    ! ---- P05 weld slots ----
    PERS bool P05W01_Used := FALSE;
    PERS num  P05W01_SubType := 0;
    PERS num  P05W01_ToolSel := 0;
    PERS num  P05W01_LenMM := 0;
    PERS robtarget P05W01_ArcStart := [[0,0,0],[1,0,0,0],[0,0,0,0],[9E9,9E9,9E9,9E9,9E9,9E9]];
    PERS robtarget P05W01_ArcEnd   := [[0,0,0],[1,0,0,0],[0,0,0,0],[9E9,9E9,9E9,9E9,9E9,9E9]];
    PERS robtarget P05W01_Approach := [[0,0,0],[1,0,0,0],[0,0,0,0],[9E9,9E9,9E9,9E9,9E9,9E9]];
    PERS robtarget P05W01_Retract  := [[0,0,0],[1,0,0,0],[0,0,0,0],[9E9,9E9,9E9,9E9,9E9,9E9]];
    PERS robtarget P05W01_Trans    := [[0,0,0],[1,0,0,0],[0,0,0,0],[9E9,9E9,9E9,9E9,9E9,9E9]];
    PERS bool P05W02_Used := FALSE;
    PERS num  P05W02_SubType := 0;
    PERS num  P05W02_ToolSel := 0;
    PERS num  P05W02_LenMM := 0;
    PERS robtarget P05W02_ArcStart := [[0,0,0],[1,0,0,0],[0,0,0,0],[9E9,9E9,9E9,9E9,9E9,9E9]];
    PERS robtarget P05W02_ArcEnd   := [[0,0,0],[1,0,0,0],[0,0,0,0],[9E9,9E9,9E9,9E9,9E9,9E9]];
    PERS robtarget P05W02_Approach := [[0,0,0],[1,0,0,0],[0,0,0,0],[9E9,9E9,9E9,9E9,9E9,9E9]];
    PERS robtarget P05W02_Retract  := [[0,0,0],[1,0,0,0],[0,0,0,0],[9E9,9E9,9E9,9E9,9E9,9E9]];
    PERS robtarget P05W02_Trans    := [[0,0,0],[1,0,0,0],[0,0,0,0],[9E9,9E9,9E9,9E9,9E9,9E9]];
    PERS bool P05W03_Used := FALSE;
    PERS num  P05W03_SubType := 0;
    PERS num  P05W03_ToolSel := 0;
    PERS num  P05W03_LenMM := 0;
    PERS robtarget P05W03_ArcStart := [[0,0,0],[1,0,0,0],[0,0,0,0],[9E9,9E9,9E9,9E9,9E9,9E9]];
    PERS robtarget P05W03_ArcEnd   := [[0,0,0],[1,0,0,0],[0,0,0,0],[9E9,9E9,9E9,9E9,9E9,9E9]];
    PERS robtarget P05W03_Approach := [[0,0,0],[1,0,0,0],[0,0,0,0],[9E9,9E9,9E9,9E9,9E9,9E9]];
    PERS robtarget P05W03_Retract  := [[0,0,0],[1,0,0,0],[0,0,0,0],[9E9,9E9,9E9,9E9,9E9,9E9]];
    PERS robtarget P05W03_Trans    := [[0,0,0],[1,0,0,0],[0,0,0,0],[9E9,9E9,9E9,9E9,9E9,9E9]];
    PERS bool P05W04_Used := FALSE;
    PERS num  P05W04_SubType := 0;
    PERS num  P05W04_ToolSel := 0;
    PERS num  P05W04_LenMM := 0;
    PERS robtarget P05W04_ArcStart := [[0,0,0],[1,0,0,0],[0,0,0,0],[9E9,9E9,9E9,9E9,9E9,9E9]];
    PERS robtarget P05W04_ArcEnd   := [[0,0,0],[1,0,0,0],[0,0,0,0],[9E9,9E9,9E9,9E9,9E9,9E9]];
    PERS robtarget P05W04_Approach := [[0,0,0],[1,0,0,0],[0,0,0,0],[9E9,9E9,9E9,9E9,9E9,9E9]];
    PERS robtarget P05W04_Retract  := [[0,0,0],[1,0,0,0],[0,0,0,0],[9E9,9E9,9E9,9E9,9E9,9E9]];
    PERS robtarget P05W04_Trans    := [[0,0,0],[1,0,0,0],[0,0,0,0],[9E9,9E9,9E9,9E9,9E9,9E9]];
    PERS bool P05W05_Used := FALSE;
    PERS num  P05W05_SubType := 0;
    PERS num  P05W05_ToolSel := 0;
    PERS num  P05W05_LenMM := 0;
    PERS robtarget P05W05_ArcStart := [[0,0,0],[1,0,0,0],[0,0,0,0],[9E9,9E9,9E9,9E9,9E9,9E9]];
    PERS robtarget P05W05_ArcEnd   := [[0,0,0],[1,0,0,0],[0,0,0,0],[9E9,9E9,9E9,9E9,9E9,9E9]];
    PERS robtarget P05W05_Approach := [[0,0,0],[1,0,0,0],[0,0,0,0],[9E9,9E9,9E9,9E9,9E9,9E9]];
    PERS robtarget P05W05_Retract  := [[0,0,0],[1,0,0,0],[0,0,0,0],[9E9,9E9,9E9,9E9,9E9,9E9]];
    PERS robtarget P05W05_Trans    := [[0,0,0],[1,0,0,0],[0,0,0,0],[9E9,9E9,9E9,9E9,9E9,9E9]];
    PERS bool P05W06_Used := FALSE;
    PERS num  P05W06_SubType := 0;
    PERS num  P05W06_ToolSel := 0;
    PERS num  P05W06_LenMM := 0;
    PERS robtarget P05W06_ArcStart := [[0,0,0],[1,0,0,0],[0,0,0,0],[9E9,9E9,9E9,9E9,9E9,9E9]];
    PERS robtarget P05W06_ArcEnd   := [[0,0,0],[1,0,0,0],[0,0,0,0],[9E9,9E9,9E9,9E9,9E9,9E9]];
    PERS robtarget P05W06_Approach := [[0,0,0],[1,0,0,0],[0,0,0,0],[9E9,9E9,9E9,9E9,9E9,9E9]];
    PERS robtarget P05W06_Retract  := [[0,0,0],[1,0,0,0],[0,0,0,0],[9E9,9E9,9E9,9E9,9E9,9E9]];
    PERS robtarget P05W06_Trans    := [[0,0,0],[1,0,0,0],[0,0,0,0],[9E9,9E9,9E9,9E9,9E9,9E9]];
    PERS bool P05W07_Used := FALSE;
    PERS num  P05W07_SubType := 0;
    PERS num  P05W07_ToolSel := 0;
    PERS num  P05W07_LenMM := 0;
    PERS robtarget P05W07_ArcStart := [[0,0,0],[1,0,0,0],[0,0,0,0],[9E9,9E9,9E9,9E9,9E9,9E9]];
    PERS robtarget P05W07_ArcEnd   := [[0,0,0],[1,0,0,0],[0,0,0,0],[9E9,9E9,9E9,9E9,9E9,9E9]];
    PERS robtarget P05W07_Approach := [[0,0,0],[1,0,0,0],[0,0,0,0],[9E9,9E9,9E9,9E9,9E9,9E9]];
    PERS robtarget P05W07_Retract  := [[0,0,0],[1,0,0,0],[0,0,0,0],[9E9,9E9,9E9,9E9,9E9,9E9]];
    PERS robtarget P05W07_Trans    := [[0,0,0],[1,0,0,0],[0,0,0,0],[9E9,9E9,9E9,9E9,9E9,9E9]];
    PERS bool P05W08_Used := FALSE;
    PERS num  P05W08_SubType := 0;
    PERS num  P05W08_ToolSel := 0;
    PERS num  P05W08_LenMM := 0;
    PERS robtarget P05W08_ArcStart := [[0,0,0],[1,0,0,0],[0,0,0,0],[9E9,9E9,9E9,9E9,9E9,9E9]];
    PERS robtarget P05W08_ArcEnd   := [[0,0,0],[1,0,0,0],[0,0,0,0],[9E9,9E9,9E9,9E9,9E9,9E9]];
    PERS robtarget P05W08_Approach := [[0,0,0],[1,0,0,0],[0,0,0,0],[9E9,9E9,9E9,9E9,9E9,9E9]];
    PERS robtarget P05W08_Retract  := [[0,0,0],[1,0,0,0],[0,0,0,0],[9E9,9E9,9E9,9E9,9E9,9E9]];
    PERS robtarget P05W08_Trans    := [[0,0,0],[1,0,0,0],[0,0,0,0],[9E9,9E9,9E9,9E9,9E9,9E9]];
    PERS bool P05W09_Used := FALSE;
    PERS num  P05W09_SubType := 0;
    PERS num  P05W09_ToolSel := 0;
    PERS num  P05W09_LenMM := 0;
    PERS robtarget P05W09_ArcStart := [[0,0,0],[1,0,0,0],[0,0,0,0],[9E9,9E9,9E9,9E9,9E9,9E9]];
    PERS robtarget P05W09_ArcEnd   := [[0,0,0],[1,0,0,0],[0,0,0,0],[9E9,9E9,9E9,9E9,9E9,9E9]];
    PERS robtarget P05W09_Approach := [[0,0,0],[1,0,0,0],[0,0,0,0],[9E9,9E9,9E9,9E9,9E9,9E9]];
    PERS robtarget P05W09_Retract  := [[0,0,0],[1,0,0,0],[0,0,0,0],[9E9,9E9,9E9,9E9,9E9,9E9]];
    PERS robtarget P05W09_Trans    := [[0,0,0],[1,0,0,0],[0,0,0,0],[9E9,9E9,9E9,9E9,9E9,9E9]];
    PERS bool P05W10_Used := FALSE;
    PERS num  P05W10_SubType := 0;
    PERS num  P05W10_ToolSel := 0;
    PERS num  P05W10_LenMM := 0;
    PERS robtarget P05W10_ArcStart := [[0,0,0],[1,0,0,0],[0,0,0,0],[9E9,9E9,9E9,9E9,9E9,9E9]];
    PERS robtarget P05W10_ArcEnd   := [[0,0,0],[1,0,0,0],[0,0,0,0],[9E9,9E9,9E9,9E9,9E9,9E9]];
    PERS robtarget P05W10_Approach := [[0,0,0],[1,0,0,0],[0,0,0,0],[9E9,9E9,9E9,9E9,9E9,9E9]];
    PERS robtarget P05W10_Retract  := [[0,0,0],[1,0,0,0],[0,0,0,0],[9E9,9E9,9E9,9E9,9E9,9E9]];
    PERS robtarget P05W10_Trans    := [[0,0,0],[1,0,0,0],[0,0,0,0],[9E9,9E9,9E9,9E9,9E9,9E9]];
    PERS bool P05W11_Used := FALSE;
    PERS num  P05W11_SubType := 0;
    PERS num  P05W11_ToolSel := 0;
    PERS num  P05W11_LenMM := 0;
    PERS robtarget P05W11_ArcStart := [[0,0,0],[1,0,0,0],[0,0,0,0],[9E9,9E9,9E9,9E9,9E9,9E9]];
    PERS robtarget P05W11_ArcEnd   := [[0,0,0],[1,0,0,0],[0,0,0,0],[9E9,9E9,9E9,9E9,9E9,9E9]];
    PERS robtarget P05W11_Approach := [[0,0,0],[1,0,0,0],[0,0,0,0],[9E9,9E9,9E9,9E9,9E9,9E9]];
    PERS robtarget P05W11_Retract  := [[0,0,0],[1,0,0,0],[0,0,0,0],[9E9,9E9,9E9,9E9,9E9,9E9]];
    PERS robtarget P05W11_Trans    := [[0,0,0],[1,0,0,0],[0,0,0,0],[9E9,9E9,9E9,9E9,9E9,9E9]];
    PERS bool P05W12_Used := FALSE;
    PERS num  P05W12_SubType := 0;
    PERS num  P05W12_ToolSel := 0;
    PERS num  P05W12_LenMM := 0;
    PERS robtarget P05W12_ArcStart := [[0,0,0],[1,0,0,0],[0,0,0,0],[9E9,9E9,9E9,9E9,9E9,9E9]];
    PERS robtarget P05W12_ArcEnd   := [[0,0,0],[1,0,0,0],[0,0,0,0],[9E9,9E9,9E9,9E9,9E9,9E9]];
    PERS robtarget P05W12_Approach := [[0,0,0],[1,0,0,0],[0,0,0,0],[9E9,9E9,9E9,9E9,9E9,9E9]];
    PERS robtarget P05W12_Retract  := [[0,0,0],[1,0,0,0],[0,0,0,0],[9E9,9E9,9E9,9E9,9E9,9E9]];
    PERS robtarget P05W12_Trans    := [[0,0,0],[1,0,0,0],[0,0,0,0],[9E9,9E9,9E9,9E9,9E9,9E9]];
    PERS bool P05W13_Used := FALSE;
    PERS num  P05W13_SubType := 0;
    PERS num  P05W13_ToolSel := 0;
    PERS num  P05W13_LenMM := 0;
    PERS robtarget P05W13_ArcStart := [[0,0,0],[1,0,0,0],[0,0,0,0],[9E9,9E9,9E9,9E9,9E9,9E9]];
    PERS robtarget P05W13_ArcEnd   := [[0,0,0],[1,0,0,0],[0,0,0,0],[9E9,9E9,9E9,9E9,9E9,9E9]];
    PERS robtarget P05W13_Approach := [[0,0,0],[1,0,0,0],[0,0,0,0],[9E9,9E9,9E9,9E9,9E9,9E9]];
    PERS robtarget P05W13_Retract  := [[0,0,0],[1,0,0,0],[0,0,0,0],[9E9,9E9,9E9,9E9,9E9,9E9]];
    PERS robtarget P05W13_Trans    := [[0,0,0],[1,0,0,0],[0,0,0,0],[9E9,9E9,9E9,9E9,9E9,9E9]];
    PERS bool P05W14_Used := FALSE;
    PERS num  P05W14_SubType := 0;
    PERS num  P05W14_ToolSel := 0;
    PERS num  P05W14_LenMM := 0;
    PERS robtarget P05W14_ArcStart := [[0,0,0],[1,0,0,0],[0,0,0,0],[9E9,9E9,9E9,9E9,9E9,9E9]];
    PERS robtarget P05W14_ArcEnd   := [[0,0,0],[1,0,0,0],[0,0,0,0],[9E9,9E9,9E9,9E9,9E9,9E9]];
    PERS robtarget P05W14_Approach := [[0,0,0],[1,0,0,0],[0,0,0,0],[9E9,9E9,9E9,9E9,9E9,9E9]];
    PERS robtarget P05W14_Retract  := [[0,0,0],[1,0,0,0],[0,0,0,0],[9E9,9E9,9E9,9E9,9E9,9E9]];
    PERS robtarget P05W14_Trans    := [[0,0,0],[1,0,0,0],[0,0,0,0],[9E9,9E9,9E9,9E9,9E9,9E9]];
    PERS bool P05W15_Used := FALSE;
    PERS num  P05W15_SubType := 0;
    PERS num  P05W15_ToolSel := 0;
    PERS num  P05W15_LenMM := 0;
    PERS robtarget P05W15_ArcStart := [[0,0,0],[1,0,0,0],[0,0,0,0],[9E9,9E9,9E9,9E9,9E9,9E9]];
    PERS robtarget P05W15_ArcEnd   := [[0,0,0],[1,0,0,0],[0,0,0,0],[9E9,9E9,9E9,9E9,9E9,9E9]];
    PERS robtarget P05W15_Approach := [[0,0,0],[1,0,0,0],[0,0,0,0],[9E9,9E9,9E9,9E9,9E9,9E9]];
    PERS robtarget P05W15_Retract  := [[0,0,0],[1,0,0,0],[0,0,0,0],[9E9,9E9,9E9,9E9,9E9,9E9]];
    PERS robtarget P05W15_Trans    := [[0,0,0],[1,0,0,0],[0,0,0,0],[9E9,9E9,9E9,9E9,9E9,9E9]];
    PERS bool P05W16_Used := FALSE;
    PERS num  P05W16_SubType := 0;
    PERS num  P05W16_ToolSel := 0;
    PERS num  P05W16_LenMM := 0;
    PERS robtarget P05W16_ArcStart := [[0,0,0],[1,0,0,0],[0,0,0,0],[9E9,9E9,9E9,9E9,9E9,9E9]];
    PERS robtarget P05W16_ArcEnd   := [[0,0,0],[1,0,0,0],[0,0,0,0],[9E9,9E9,9E9,9E9,9E9,9E9]];
    PERS robtarget P05W16_Approach := [[0,0,0],[1,0,0,0],[0,0,0,0],[9E9,9E9,9E9,9E9,9E9,9E9]];
    PERS robtarget P05W16_Retract  := [[0,0,0],[1,0,0,0],[0,0,0,0],[9E9,9E9,9E9,9E9,9E9,9E9]];
    PERS robtarget P05W16_Trans    := [[0,0,0],[1,0,0,0],[0,0,0,0],[9E9,9E9,9E9,9E9,9E9,9E9]];
    PERS bool P05W17_Used := FALSE;
    PERS num  P05W17_SubType := 0;
    PERS num  P05W17_ToolSel := 0;
    PERS num  P05W17_LenMM := 0;
    PERS robtarget P05W17_ArcStart := [[0,0,0],[1,0,0,0],[0,0,0,0],[9E9,9E9,9E9,9E9,9E9,9E9]];
    PERS robtarget P05W17_ArcEnd   := [[0,0,0],[1,0,0,0],[0,0,0,0],[9E9,9E9,9E9,9E9,9E9,9E9]];
    PERS robtarget P05W17_Approach := [[0,0,0],[1,0,0,0],[0,0,0,0],[9E9,9E9,9E9,9E9,9E9,9E9]];
    PERS robtarget P05W17_Retract  := [[0,0,0],[1,0,0,0],[0,0,0,0],[9E9,9E9,9E9,9E9,9E9,9E9]];
    PERS robtarget P05W17_Trans    := [[0,0,0],[1,0,0,0],[0,0,0,0],[9E9,9E9,9E9,9E9,9E9,9E9]];
    PERS bool P05W18_Used := FALSE;
    PERS num  P05W18_SubType := 0;
    PERS num  P05W18_ToolSel := 0;
    PERS num  P05W18_LenMM := 0;
    PERS robtarget P05W18_ArcStart := [[0,0,0],[1,0,0,0],[0,0,0,0],[9E9,9E9,9E9,9E9,9E9,9E9]];
    PERS robtarget P05W18_ArcEnd   := [[0,0,0],[1,0,0,0],[0,0,0,0],[9E9,9E9,9E9,9E9,9E9,9E9]];
    PERS robtarget P05W18_Approach := [[0,0,0],[1,0,0,0],[0,0,0,0],[9E9,9E9,9E9,9E9,9E9,9E9]];
    PERS robtarget P05W18_Retract  := [[0,0,0],[1,0,0,0],[0,0,0,0],[9E9,9E9,9E9,9E9,9E9,9E9]];
    PERS robtarget P05W18_Trans    := [[0,0,0],[1,0,0,0],[0,0,0,0],[9E9,9E9,9E9,9E9,9E9,9E9]];
    PERS bool P05W19_Used := FALSE;
    PERS num  P05W19_SubType := 0;
    PERS num  P05W19_ToolSel := 0;
    PERS num  P05W19_LenMM := 0;
    PERS robtarget P05W19_ArcStart := [[0,0,0],[1,0,0,0],[0,0,0,0],[9E9,9E9,9E9,9E9,9E9,9E9]];
    PERS robtarget P05W19_ArcEnd   := [[0,0,0],[1,0,0,0],[0,0,0,0],[9E9,9E9,9E9,9E9,9E9,9E9]];
    PERS robtarget P05W19_Approach := [[0,0,0],[1,0,0,0],[0,0,0,0],[9E9,9E9,9E9,9E9,9E9,9E9]];
    PERS robtarget P05W19_Retract  := [[0,0,0],[1,0,0,0],[0,0,0,0],[9E9,9E9,9E9,9E9,9E9,9E9]];
    PERS robtarget P05W19_Trans    := [[0,0,0],[1,0,0,0],[0,0,0,0],[9E9,9E9,9E9,9E9,9E9,9E9]];
    PERS bool P05W20_Used := FALSE;
    PERS num  P05W20_SubType := 0;
    PERS num  P05W20_ToolSel := 0;
    PERS num  P05W20_LenMM := 0;
    PERS robtarget P05W20_ArcStart := [[0,0,0],[1,0,0,0],[0,0,0,0],[9E9,9E9,9E9,9E9,9E9,9E9]];
    PERS robtarget P05W20_ArcEnd   := [[0,0,0],[1,0,0,0],[0,0,0,0],[9E9,9E9,9E9,9E9,9E9,9E9]];
    PERS robtarget P05W20_Approach := [[0,0,0],[1,0,0,0],[0,0,0,0],[9E9,9E9,9E9,9E9,9E9,9E9]];
    PERS robtarget P05W20_Retract  := [[0,0,0],[1,0,0,0],[0,0,0,0],[9E9,9E9,9E9,9E9,9E9,9E9]];
    PERS robtarget P05W20_Trans    := [[0,0,0],[1,0,0,0],[0,0,0,0],[9E9,9E9,9E9,9E9,9E9,9E9]];
    PERS bool P05W21_Used := FALSE;
    PERS num  P05W21_SubType := 0;
    PERS num  P05W21_ToolSel := 0;
    PERS num  P05W21_LenMM := 0;
    PERS robtarget P05W21_ArcStart := [[0,0,0],[1,0,0,0],[0,0,0,0],[9E9,9E9,9E9,9E9,9E9,9E9]];
    PERS robtarget P05W21_ArcEnd   := [[0,0,0],[1,0,0,0],[0,0,0,0],[9E9,9E9,9E9,9E9,9E9,9E9]];
    PERS robtarget P05W21_Approach := [[0,0,0],[1,0,0,0],[0,0,0,0],[9E9,9E9,9E9,9E9,9E9,9E9]];
    PERS robtarget P05W21_Retract  := [[0,0,0],[1,0,0,0],[0,0,0,0],[9E9,9E9,9E9,9E9,9E9,9E9]];
    PERS robtarget P05W21_Trans    := [[0,0,0],[1,0,0,0],[0,0,0,0],[9E9,9E9,9E9,9E9,9E9,9E9]];
    PERS bool P05W22_Used := FALSE;
    PERS num  P05W22_SubType := 0;
    PERS num  P05W22_ToolSel := 0;
    PERS num  P05W22_LenMM := 0;
    PERS robtarget P05W22_ArcStart := [[0,0,0],[1,0,0,0],[0,0,0,0],[9E9,9E9,9E9,9E9,9E9,9E9]];
    PERS robtarget P05W22_ArcEnd   := [[0,0,0],[1,0,0,0],[0,0,0,0],[9E9,9E9,9E9,9E9,9E9,9E9]];
    PERS robtarget P05W22_Approach := [[0,0,0],[1,0,0,0],[0,0,0,0],[9E9,9E9,9E9,9E9,9E9,9E9]];
    PERS robtarget P05W22_Retract  := [[0,0,0],[1,0,0,0],[0,0,0,0],[9E9,9E9,9E9,9E9,9E9,9E9]];
    PERS robtarget P05W22_Trans    := [[0,0,0],[1,0,0,0],[0,0,0,0],[9E9,9E9,9E9,9E9,9E9,9E9]];
    PERS bool P05W23_Used := FALSE;
    PERS num  P05W23_SubType := 0;
    PERS num  P05W23_ToolSel := 0;
    PERS num  P05W23_LenMM := 0;
    PERS robtarget P05W23_ArcStart := [[0,0,0],[1,0,0,0],[0,0,0,0],[9E9,9E9,9E9,9E9,9E9,9E9]];
    PERS robtarget P05W23_ArcEnd   := [[0,0,0],[1,0,0,0],[0,0,0,0],[9E9,9E9,9E9,9E9,9E9,9E9]];
    PERS robtarget P05W23_Approach := [[0,0,0],[1,0,0,0],[0,0,0,0],[9E9,9E9,9E9,9E9,9E9,9E9]];
    PERS robtarget P05W23_Retract  := [[0,0,0],[1,0,0,0],[0,0,0,0],[9E9,9E9,9E9,9E9,9E9,9E9]];
    PERS robtarget P05W23_Trans    := [[0,0,0],[1,0,0,0],[0,0,0,0],[9E9,9E9,9E9,9E9,9E9,9E9]];
    PERS bool P05W24_Used := FALSE;
    PERS num  P05W24_SubType := 0;
    PERS num  P05W24_ToolSel := 0;
    PERS num  P05W24_LenMM := 0;
    PERS robtarget P05W24_ArcStart := [[0,0,0],[1,0,0,0],[0,0,0,0],[9E9,9E9,9E9,9E9,9E9,9E9]];
    PERS robtarget P05W24_ArcEnd   := [[0,0,0],[1,0,0,0],[0,0,0,0],[9E9,9E9,9E9,9E9,9E9,9E9]];
    PERS robtarget P05W24_Approach := [[0,0,0],[1,0,0,0],[0,0,0,0],[9E9,9E9,9E9,9E9,9E9,9E9]];
    PERS robtarget P05W24_Retract  := [[0,0,0],[1,0,0,0],[0,0,0,0],[9E9,9E9,9E9,9E9,9E9,9E9]];
    PERS robtarget P05W24_Trans    := [[0,0,0],[1,0,0,0],[0,0,0,0],[9E9,9E9,9E9,9E9,9E9,9E9]];
    PERS bool P05W25_Used := FALSE;
    PERS num  P05W25_SubType := 0;
    PERS num  P05W25_ToolSel := 0;
    PERS num  P05W25_LenMM := 0;
    PERS robtarget P05W25_ArcStart := [[0,0,0],[1,0,0,0],[0,0,0,0],[9E9,9E9,9E9,9E9,9E9,9E9]];
    PERS robtarget P05W25_ArcEnd   := [[0,0,0],[1,0,0,0],[0,0,0,0],[9E9,9E9,9E9,9E9,9E9,9E9]];
    PERS robtarget P05W25_Approach := [[0,0,0],[1,0,0,0],[0,0,0,0],[9E9,9E9,9E9,9E9,9E9,9E9]];
    PERS robtarget P05W25_Retract  := [[0,0,0],[1,0,0,0],[0,0,0,0],[9E9,9E9,9E9,9E9,9E9,9E9]];
    PERS robtarget P05W25_Trans    := [[0,0,0],[1,0,0,0],[0,0,0,0],[9E9,9E9,9E9,9E9,9E9,9E9]];
    PERS bool P05W26_Used := FALSE;
    PERS num  P05W26_SubType := 0;
    PERS num  P05W26_ToolSel := 0;
    PERS num  P05W26_LenMM := 0;
    PERS robtarget P05W26_ArcStart := [[0,0,0],[1,0,0,0],[0,0,0,0],[9E9,9E9,9E9,9E9,9E9,9E9]];
    PERS robtarget P05W26_ArcEnd   := [[0,0,0],[1,0,0,0],[0,0,0,0],[9E9,9E9,9E9,9E9,9E9,9E9]];
    PERS robtarget P05W26_Approach := [[0,0,0],[1,0,0,0],[0,0,0,0],[9E9,9E9,9E9,9E9,9E9,9E9]];
    PERS robtarget P05W26_Retract  := [[0,0,0],[1,0,0,0],[0,0,0,0],[9E9,9E9,9E9,9E9,9E9,9E9]];
    PERS robtarget P05W26_Trans    := [[0,0,0],[1,0,0,0],[0,0,0,0],[9E9,9E9,9E9,9E9,9E9,9E9]];
    PERS bool P05W27_Used := FALSE;
    PERS num  P05W27_SubType := 0;
    PERS num  P05W27_ToolSel := 0;
    PERS num  P05W27_LenMM := 0;
    PERS robtarget P05W27_ArcStart := [[0,0,0],[1,0,0,0],[0,0,0,0],[9E9,9E9,9E9,9E9,9E9,9E9]];
    PERS robtarget P05W27_ArcEnd   := [[0,0,0],[1,0,0,0],[0,0,0,0],[9E9,9E9,9E9,9E9,9E9,9E9]];
    PERS robtarget P05W27_Approach := [[0,0,0],[1,0,0,0],[0,0,0,0],[9E9,9E9,9E9,9E9,9E9,9E9]];
    PERS robtarget P05W27_Retract  := [[0,0,0],[1,0,0,0],[0,0,0,0],[9E9,9E9,9E9,9E9,9E9,9E9]];
    PERS robtarget P05W27_Trans    := [[0,0,0],[1,0,0,0],[0,0,0,0],[9E9,9E9,9E9,9E9,9E9,9E9]];
    PERS bool P05W28_Used := FALSE;
    PERS num  P05W28_SubType := 0;
    PERS num  P05W28_ToolSel := 0;
    PERS num  P05W28_LenMM := 0;
    PERS robtarget P05W28_ArcStart := [[0,0,0],[1,0,0,0],[0,0,0,0],[9E9,9E9,9E9,9E9,9E9,9E9]];
    PERS robtarget P05W28_ArcEnd   := [[0,0,0],[1,0,0,0],[0,0,0,0],[9E9,9E9,9E9,9E9,9E9,9E9]];
    PERS robtarget P05W28_Approach := [[0,0,0],[1,0,0,0],[0,0,0,0],[9E9,9E9,9E9,9E9,9E9,9E9]];
    PERS robtarget P05W28_Retract  := [[0,0,0],[1,0,0,0],[0,0,0,0],[9E9,9E9,9E9,9E9,9E9,9E9]];
    PERS robtarget P05W28_Trans    := [[0,0,0],[1,0,0,0],[0,0,0,0],[9E9,9E9,9E9,9E9,9E9,9E9]];
    PERS bool P05W29_Used := FALSE;
    PERS num  P05W29_SubType := 0;
    PERS num  P05W29_ToolSel := 0;
    PERS num  P05W29_LenMM := 0;
    PERS robtarget P05W29_ArcStart := [[0,0,0],[1,0,0,0],[0,0,0,0],[9E9,9E9,9E9,9E9,9E9,9E9]];
    PERS robtarget P05W29_ArcEnd   := [[0,0,0],[1,0,0,0],[0,0,0,0],[9E9,9E9,9E9,9E9,9E9,9E9]];
    PERS robtarget P05W29_Approach := [[0,0,0],[1,0,0,0],[0,0,0,0],[9E9,9E9,9E9,9E9,9E9,9E9]];
    PERS robtarget P05W29_Retract  := [[0,0,0],[1,0,0,0],[0,0,0,0],[9E9,9E9,9E9,9E9,9E9,9E9]];
    PERS robtarget P05W29_Trans    := [[0,0,0],[1,0,0,0],[0,0,0,0],[9E9,9E9,9E9,9E9,9E9,9E9]];
    PERS bool P05W30_Used := FALSE;
    PERS num  P05W30_SubType := 0;
    PERS num  P05W30_ToolSel := 0;
    PERS num  P05W30_LenMM := 0;
    PERS robtarget P05W30_ArcStart := [[0,0,0],[1,0,0,0],[0,0,0,0],[9E9,9E9,9E9,9E9,9E9,9E9]];
    PERS robtarget P05W30_ArcEnd   := [[0,0,0],[1,0,0,0],[0,0,0,0],[9E9,9E9,9E9,9E9,9E9,9E9]];
    PERS robtarget P05W30_Approach := [[0,0,0],[1,0,0,0],[0,0,0,0],[9E9,9E9,9E9,9E9,9E9,9E9]];
    PERS robtarget P05W30_Retract  := [[0,0,0],[1,0,0,0],[0,0,0,0],[9E9,9E9,9E9,9E9,9E9,9E9]];
    PERS robtarget P05W30_Trans    := [[0,0,0],[1,0,0,0],[0,0,0,0],[9E9,9E9,9E9,9E9,9E9,9E9]];

    ! ---- P06 weld slots ----
    PERS bool P06W01_Used := FALSE;
    PERS num  P06W01_SubType := 0;
    PERS num  P06W01_ToolSel := 0;
    PERS num  P06W01_LenMM := 0;
    PERS robtarget P06W01_ArcStart := [[0,0,0],[1,0,0,0],[0,0,0,0],[9E9,9E9,9E9,9E9,9E9,9E9]];
    PERS robtarget P06W01_ArcEnd   := [[0,0,0],[1,0,0,0],[0,0,0,0],[9E9,9E9,9E9,9E9,9E9,9E9]];
    PERS robtarget P06W01_Approach := [[0,0,0],[1,0,0,0],[0,0,0,0],[9E9,9E9,9E9,9E9,9E9,9E9]];
    PERS robtarget P06W01_Retract  := [[0,0,0],[1,0,0,0],[0,0,0,0],[9E9,9E9,9E9,9E9,9E9,9E9]];
    PERS robtarget P06W01_Trans    := [[0,0,0],[1,0,0,0],[0,0,0,0],[9E9,9E9,9E9,9E9,9E9,9E9]];
    PERS bool P06W02_Used := FALSE;
    PERS num  P06W02_SubType := 0;
    PERS num  P06W02_ToolSel := 0;
    PERS num  P06W02_LenMM := 0;
    PERS robtarget P06W02_ArcStart := [[0,0,0],[1,0,0,0],[0,0,0,0],[9E9,9E9,9E9,9E9,9E9,9E9]];
    PERS robtarget P06W02_ArcEnd   := [[0,0,0],[1,0,0,0],[0,0,0,0],[9E9,9E9,9E9,9E9,9E9,9E9]];
    PERS robtarget P06W02_Approach := [[0,0,0],[1,0,0,0],[0,0,0,0],[9E9,9E9,9E9,9E9,9E9,9E9]];
    PERS robtarget P06W02_Retract  := [[0,0,0],[1,0,0,0],[0,0,0,0],[9E9,9E9,9E9,9E9,9E9,9E9]];
    PERS robtarget P06W02_Trans    := [[0,0,0],[1,0,0,0],[0,0,0,0],[9E9,9E9,9E9,9E9,9E9,9E9]];
    PERS bool P06W03_Used := FALSE;
    PERS num  P06W03_SubType := 0;
    PERS num  P06W03_ToolSel := 0;
    PERS num  P06W03_LenMM := 0;
    PERS robtarget P06W03_ArcStart := [[0,0,0],[1,0,0,0],[0,0,0,0],[9E9,9E9,9E9,9E9,9E9,9E9]];
    PERS robtarget P06W03_ArcEnd   := [[0,0,0],[1,0,0,0],[0,0,0,0],[9E9,9E9,9E9,9E9,9E9,9E9]];
    PERS robtarget P06W03_Approach := [[0,0,0],[1,0,0,0],[0,0,0,0],[9E9,9E9,9E9,9E9,9E9,9E9]];
    PERS robtarget P06W03_Retract  := [[0,0,0],[1,0,0,0],[0,0,0,0],[9E9,9E9,9E9,9E9,9E9,9E9]];
    PERS robtarget P06W03_Trans    := [[0,0,0],[1,0,0,0],[0,0,0,0],[9E9,9E9,9E9,9E9,9E9,9E9]];
    PERS bool P06W04_Used := FALSE;
    PERS num  P06W04_SubType := 0;
    PERS num  P06W04_ToolSel := 0;
    PERS num  P06W04_LenMM := 0;
    PERS robtarget P06W04_ArcStart := [[0,0,0],[1,0,0,0],[0,0,0,0],[9E9,9E9,9E9,9E9,9E9,9E9]];
    PERS robtarget P06W04_ArcEnd   := [[0,0,0],[1,0,0,0],[0,0,0,0],[9E9,9E9,9E9,9E9,9E9,9E9]];
    PERS robtarget P06W04_Approach := [[0,0,0],[1,0,0,0],[0,0,0,0],[9E9,9E9,9E9,9E9,9E9,9E9]];
    PERS robtarget P06W04_Retract  := [[0,0,0],[1,0,0,0],[0,0,0,0],[9E9,9E9,9E9,9E9,9E9,9E9]];
    PERS robtarget P06W04_Trans    := [[0,0,0],[1,0,0,0],[0,0,0,0],[9E9,9E9,9E9,9E9,9E9,9E9]];
    PERS bool P06W05_Used := FALSE;
    PERS num  P06W05_SubType := 0;
    PERS num  P06W05_ToolSel := 0;
    PERS num  P06W05_LenMM := 0;
    PERS robtarget P06W05_ArcStart := [[0,0,0],[1,0,0,0],[0,0,0,0],[9E9,9E9,9E9,9E9,9E9,9E9]];
    PERS robtarget P06W05_ArcEnd   := [[0,0,0],[1,0,0,0],[0,0,0,0],[9E9,9E9,9E9,9E9,9E9,9E9]];
    PERS robtarget P06W05_Approach := [[0,0,0],[1,0,0,0],[0,0,0,0],[9E9,9E9,9E9,9E9,9E9,9E9]];
    PERS robtarget P06W05_Retract  := [[0,0,0],[1,0,0,0],[0,0,0,0],[9E9,9E9,9E9,9E9,9E9,9E9]];
    PERS robtarget P06W05_Trans    := [[0,0,0],[1,0,0,0],[0,0,0,0],[9E9,9E9,9E9,9E9,9E9,9E9]];
    PERS bool P06W06_Used := FALSE;
    PERS num  P06W06_SubType := 0;
    PERS num  P06W06_ToolSel := 0;
    PERS num  P06W06_LenMM := 0;
    PERS robtarget P06W06_ArcStart := [[0,0,0],[1,0,0,0],[0,0,0,0],[9E9,9E9,9E9,9E9,9E9,9E9]];
    PERS robtarget P06W06_ArcEnd   := [[0,0,0],[1,0,0,0],[0,0,0,0],[9E9,9E9,9E9,9E9,9E9,9E9]];
    PERS robtarget P06W06_Approach := [[0,0,0],[1,0,0,0],[0,0,0,0],[9E9,9E9,9E9,9E9,9E9,9E9]];
    PERS robtarget P06W06_Retract  := [[0,0,0],[1,0,0,0],[0,0,0,0],[9E9,9E9,9E9,9E9,9E9,9E9]];
    PERS robtarget P06W06_Trans    := [[0,0,0],[1,0,0,0],[0,0,0,0],[9E9,9E9,9E9,9E9,9E9,9E9]];
    PERS bool P06W07_Used := FALSE;
    PERS num  P06W07_SubType := 0;
    PERS num  P06W07_ToolSel := 0;
    PERS num  P06W07_LenMM := 0;
    PERS robtarget P06W07_ArcStart := [[0,0,0],[1,0,0,0],[0,0,0,0],[9E9,9E9,9E9,9E9,9E9,9E9]];
    PERS robtarget P06W07_ArcEnd   := [[0,0,0],[1,0,0,0],[0,0,0,0],[9E9,9E9,9E9,9E9,9E9,9E9]];
    PERS robtarget P06W07_Approach := [[0,0,0],[1,0,0,0],[0,0,0,0],[9E9,9E9,9E9,9E9,9E9,9E9]];
    PERS robtarget P06W07_Retract  := [[0,0,0],[1,0,0,0],[0,0,0,0],[9E9,9E9,9E9,9E9,9E9,9E9]];
    PERS robtarget P06W07_Trans    := [[0,0,0],[1,0,0,0],[0,0,0,0],[9E9,9E9,9E9,9E9,9E9,9E9]];
    PERS bool P06W08_Used := FALSE;
    PERS num  P06W08_SubType := 0;
    PERS num  P06W08_ToolSel := 0;
    PERS num  P06W08_LenMM := 0;
    PERS robtarget P06W08_ArcStart := [[0,0,0],[1,0,0,0],[0,0,0,0],[9E9,9E9,9E9,9E9,9E9,9E9]];
    PERS robtarget P06W08_ArcEnd   := [[0,0,0],[1,0,0,0],[0,0,0,0],[9E9,9E9,9E9,9E9,9E9,9E9]];
    PERS robtarget P06W08_Approach := [[0,0,0],[1,0,0,0],[0,0,0,0],[9E9,9E9,9E9,9E9,9E9,9E9]];
    PERS robtarget P06W08_Retract  := [[0,0,0],[1,0,0,0],[0,0,0,0],[9E9,9E9,9E9,9E9,9E9,9E9]];
    PERS robtarget P06W08_Trans    := [[0,0,0],[1,0,0,0],[0,0,0,0],[9E9,9E9,9E9,9E9,9E9,9E9]];
    PERS bool P06W09_Used := FALSE;
    PERS num  P06W09_SubType := 0;
    PERS num  P06W09_ToolSel := 0;
    PERS num  P06W09_LenMM := 0;
    PERS robtarget P06W09_ArcStart := [[0,0,0],[1,0,0,0],[0,0,0,0],[9E9,9E9,9E9,9E9,9E9,9E9]];
    PERS robtarget P06W09_ArcEnd   := [[0,0,0],[1,0,0,0],[0,0,0,0],[9E9,9E9,9E9,9E9,9E9,9E9]];
    PERS robtarget P06W09_Approach := [[0,0,0],[1,0,0,0],[0,0,0,0],[9E9,9E9,9E9,9E9,9E9,9E9]];
    PERS robtarget P06W09_Retract  := [[0,0,0],[1,0,0,0],[0,0,0,0],[9E9,9E9,9E9,9E9,9E9,9E9]];
    PERS robtarget P06W09_Trans    := [[0,0,0],[1,0,0,0],[0,0,0,0],[9E9,9E9,9E9,9E9,9E9,9E9]];
    PERS bool P06W10_Used := FALSE;
    PERS num  P06W10_SubType := 0;
    PERS num  P06W10_ToolSel := 0;
    PERS num  P06W10_LenMM := 0;
    PERS robtarget P06W10_ArcStart := [[0,0,0],[1,0,0,0],[0,0,0,0],[9E9,9E9,9E9,9E9,9E9,9E9]];
    PERS robtarget P06W10_ArcEnd   := [[0,0,0],[1,0,0,0],[0,0,0,0],[9E9,9E9,9E9,9E9,9E9,9E9]];
    PERS robtarget P06W10_Approach := [[0,0,0],[1,0,0,0],[0,0,0,0],[9E9,9E9,9E9,9E9,9E9,9E9]];
    PERS robtarget P06W10_Retract  := [[0,0,0],[1,0,0,0],[0,0,0,0],[9E9,9E9,9E9,9E9,9E9,9E9]];
    PERS robtarget P06W10_Trans    := [[0,0,0],[1,0,0,0],[0,0,0,0],[9E9,9E9,9E9,9E9,9E9,9E9]];
    PERS bool P06W11_Used := FALSE;
    PERS num  P06W11_SubType := 0;
    PERS num  P06W11_ToolSel := 0;
    PERS num  P06W11_LenMM := 0;
    PERS robtarget P06W11_ArcStart := [[0,0,0],[1,0,0,0],[0,0,0,0],[9E9,9E9,9E9,9E9,9E9,9E9]];
    PERS robtarget P06W11_ArcEnd   := [[0,0,0],[1,0,0,0],[0,0,0,0],[9E9,9E9,9E9,9E9,9E9,9E9]];
    PERS robtarget P06W11_Approach := [[0,0,0],[1,0,0,0],[0,0,0,0],[9E9,9E9,9E9,9E9,9E9,9E9]];
    PERS robtarget P06W11_Retract  := [[0,0,0],[1,0,0,0],[0,0,0,0],[9E9,9E9,9E9,9E9,9E9,9E9]];
    PERS robtarget P06W11_Trans    := [[0,0,0],[1,0,0,0],[0,0,0,0],[9E9,9E9,9E9,9E9,9E9,9E9]];
    PERS bool P06W12_Used := FALSE;
    PERS num  P06W12_SubType := 0;
    PERS num  P06W12_ToolSel := 0;
    PERS num  P06W12_LenMM := 0;
    PERS robtarget P06W12_ArcStart := [[0,0,0],[1,0,0,0],[0,0,0,0],[9E9,9E9,9E9,9E9,9E9,9E9]];
    PERS robtarget P06W12_ArcEnd   := [[0,0,0],[1,0,0,0],[0,0,0,0],[9E9,9E9,9E9,9E9,9E9,9E9]];
    PERS robtarget P06W12_Approach := [[0,0,0],[1,0,0,0],[0,0,0,0],[9E9,9E9,9E9,9E9,9E9,9E9]];
    PERS robtarget P06W12_Retract  := [[0,0,0],[1,0,0,0],[0,0,0,0],[9E9,9E9,9E9,9E9,9E9,9E9]];
    PERS robtarget P06W12_Trans    := [[0,0,0],[1,0,0,0],[0,0,0,0],[9E9,9E9,9E9,9E9,9E9,9E9]];
    PERS bool P06W13_Used := FALSE;
    PERS num  P06W13_SubType := 0;
    PERS num  P06W13_ToolSel := 0;
    PERS num  P06W13_LenMM := 0;
    PERS robtarget P06W13_ArcStart := [[0,0,0],[1,0,0,0],[0,0,0,0],[9E9,9E9,9E9,9E9,9E9,9E9]];
    PERS robtarget P06W13_ArcEnd   := [[0,0,0],[1,0,0,0],[0,0,0,0],[9E9,9E9,9E9,9E9,9E9,9E9]];
    PERS robtarget P06W13_Approach := [[0,0,0],[1,0,0,0],[0,0,0,0],[9E9,9E9,9E9,9E9,9E9,9E9]];
    PERS robtarget P06W13_Retract  := [[0,0,0],[1,0,0,0],[0,0,0,0],[9E9,9E9,9E9,9E9,9E9,9E9]];
    PERS robtarget P06W13_Trans    := [[0,0,0],[1,0,0,0],[0,0,0,0],[9E9,9E9,9E9,9E9,9E9,9E9]];
    PERS bool P06W14_Used := FALSE;
    PERS num  P06W14_SubType := 0;
    PERS num  P06W14_ToolSel := 0;
    PERS num  P06W14_LenMM := 0;
    PERS robtarget P06W14_ArcStart := [[0,0,0],[1,0,0,0],[0,0,0,0],[9E9,9E9,9E9,9E9,9E9,9E9]];
    PERS robtarget P06W14_ArcEnd   := [[0,0,0],[1,0,0,0],[0,0,0,0],[9E9,9E9,9E9,9E9,9E9,9E9]];
    PERS robtarget P06W14_Approach := [[0,0,0],[1,0,0,0],[0,0,0,0],[9E9,9E9,9E9,9E9,9E9,9E9]];
    PERS robtarget P06W14_Retract  := [[0,0,0],[1,0,0,0],[0,0,0,0],[9E9,9E9,9E9,9E9,9E9,9E9]];
    PERS robtarget P06W14_Trans    := [[0,0,0],[1,0,0,0],[0,0,0,0],[9E9,9E9,9E9,9E9,9E9,9E9]];
    PERS bool P06W15_Used := FALSE;
    PERS num  P06W15_SubType := 0;
    PERS num  P06W15_ToolSel := 0;
    PERS num  P06W15_LenMM := 0;
    PERS robtarget P06W15_ArcStart := [[0,0,0],[1,0,0,0],[0,0,0,0],[9E9,9E9,9E9,9E9,9E9,9E9]];
    PERS robtarget P06W15_ArcEnd   := [[0,0,0],[1,0,0,0],[0,0,0,0],[9E9,9E9,9E9,9E9,9E9,9E9]];
    PERS robtarget P06W15_Approach := [[0,0,0],[1,0,0,0],[0,0,0,0],[9E9,9E9,9E9,9E9,9E9,9E9]];
    PERS robtarget P06W15_Retract  := [[0,0,0],[1,0,0,0],[0,0,0,0],[9E9,9E9,9E9,9E9,9E9,9E9]];
    PERS robtarget P06W15_Trans    := [[0,0,0],[1,0,0,0],[0,0,0,0],[9E9,9E9,9E9,9E9,9E9,9E9]];
    PERS bool P06W16_Used := FALSE;
    PERS num  P06W16_SubType := 0;
    PERS num  P06W16_ToolSel := 0;
    PERS num  P06W16_LenMM := 0;
    PERS robtarget P06W16_ArcStart := [[0,0,0],[1,0,0,0],[0,0,0,0],[9E9,9E9,9E9,9E9,9E9,9E9]];
    PERS robtarget P06W16_ArcEnd   := [[0,0,0],[1,0,0,0],[0,0,0,0],[9E9,9E9,9E9,9E9,9E9,9E9]];
    PERS robtarget P06W16_Approach := [[0,0,0],[1,0,0,0],[0,0,0,0],[9E9,9E9,9E9,9E9,9E9,9E9]];
    PERS robtarget P06W16_Retract  := [[0,0,0],[1,0,0,0],[0,0,0,0],[9E9,9E9,9E9,9E9,9E9,9E9]];
    PERS robtarget P06W16_Trans    := [[0,0,0],[1,0,0,0],[0,0,0,0],[9E9,9E9,9E9,9E9,9E9,9E9]];
    PERS bool P06W17_Used := FALSE;
    PERS num  P06W17_SubType := 0;
    PERS num  P06W17_ToolSel := 0;
    PERS num  P06W17_LenMM := 0;
    PERS robtarget P06W17_ArcStart := [[0,0,0],[1,0,0,0],[0,0,0,0],[9E9,9E9,9E9,9E9,9E9,9E9]];
    PERS robtarget P06W17_ArcEnd   := [[0,0,0],[1,0,0,0],[0,0,0,0],[9E9,9E9,9E9,9E9,9E9,9E9]];
    PERS robtarget P06W17_Approach := [[0,0,0],[1,0,0,0],[0,0,0,0],[9E9,9E9,9E9,9E9,9E9,9E9]];
    PERS robtarget P06W17_Retract  := [[0,0,0],[1,0,0,0],[0,0,0,0],[9E9,9E9,9E9,9E9,9E9,9E9]];
    PERS robtarget P06W17_Trans    := [[0,0,0],[1,0,0,0],[0,0,0,0],[9E9,9E9,9E9,9E9,9E9,9E9]];
    PERS bool P06W18_Used := FALSE;
    PERS num  P06W18_SubType := 0;
    PERS num  P06W18_ToolSel := 0;
    PERS num  P06W18_LenMM := 0;
    PERS robtarget P06W18_ArcStart := [[0,0,0],[1,0,0,0],[0,0,0,0],[9E9,9E9,9E9,9E9,9E9,9E9]];
    PERS robtarget P06W18_ArcEnd   := [[0,0,0],[1,0,0,0],[0,0,0,0],[9E9,9E9,9E9,9E9,9E9,9E9]];
    PERS robtarget P06W18_Approach := [[0,0,0],[1,0,0,0],[0,0,0,0],[9E9,9E9,9E9,9E9,9E9,9E9]];
    PERS robtarget P06W18_Retract  := [[0,0,0],[1,0,0,0],[0,0,0,0],[9E9,9E9,9E9,9E9,9E9,9E9]];
    PERS robtarget P06W18_Trans    := [[0,0,0],[1,0,0,0],[0,0,0,0],[9E9,9E9,9E9,9E9,9E9,9E9]];
    PERS bool P06W19_Used := FALSE;
    PERS num  P06W19_SubType := 0;
    PERS num  P06W19_ToolSel := 0;
    PERS num  P06W19_LenMM := 0;
    PERS robtarget P06W19_ArcStart := [[0,0,0],[1,0,0,0],[0,0,0,0],[9E9,9E9,9E9,9E9,9E9,9E9]];
    PERS robtarget P06W19_ArcEnd   := [[0,0,0],[1,0,0,0],[0,0,0,0],[9E9,9E9,9E9,9E9,9E9,9E9]];
    PERS robtarget P06W19_Approach := [[0,0,0],[1,0,0,0],[0,0,0,0],[9E9,9E9,9E9,9E9,9E9,9E9]];
    PERS robtarget P06W19_Retract  := [[0,0,0],[1,0,0,0],[0,0,0,0],[9E9,9E9,9E9,9E9,9E9,9E9]];
    PERS robtarget P06W19_Trans    := [[0,0,0],[1,0,0,0],[0,0,0,0],[9E9,9E9,9E9,9E9,9E9,9E9]];
    PERS bool P06W20_Used := FALSE;
    PERS num  P06W20_SubType := 0;
    PERS num  P06W20_ToolSel := 0;
    PERS num  P06W20_LenMM := 0;
    PERS robtarget P06W20_ArcStart := [[0,0,0],[1,0,0,0],[0,0,0,0],[9E9,9E9,9E9,9E9,9E9,9E9]];
    PERS robtarget P06W20_ArcEnd   := [[0,0,0],[1,0,0,0],[0,0,0,0],[9E9,9E9,9E9,9E9,9E9,9E9]];
    PERS robtarget P06W20_Approach := [[0,0,0],[1,0,0,0],[0,0,0,0],[9E9,9E9,9E9,9E9,9E9,9E9]];
    PERS robtarget P06W20_Retract  := [[0,0,0],[1,0,0,0],[0,0,0,0],[9E9,9E9,9E9,9E9,9E9,9E9]];
    PERS robtarget P06W20_Trans    := [[0,0,0],[1,0,0,0],[0,0,0,0],[9E9,9E9,9E9,9E9,9E9,9E9]];
    PERS bool P06W21_Used := FALSE;
    PERS num  P06W21_SubType := 0;
    PERS num  P06W21_ToolSel := 0;
    PERS num  P06W21_LenMM := 0;
    PERS robtarget P06W21_ArcStart := [[0,0,0],[1,0,0,0],[0,0,0,0],[9E9,9E9,9E9,9E9,9E9,9E9]];
    PERS robtarget P06W21_ArcEnd   := [[0,0,0],[1,0,0,0],[0,0,0,0],[9E9,9E9,9E9,9E9,9E9,9E9]];
    PERS robtarget P06W21_Approach := [[0,0,0],[1,0,0,0],[0,0,0,0],[9E9,9E9,9E9,9E9,9E9,9E9]];
    PERS robtarget P06W21_Retract  := [[0,0,0],[1,0,0,0],[0,0,0,0],[9E9,9E9,9E9,9E9,9E9,9E9]];
    PERS robtarget P06W21_Trans    := [[0,0,0],[1,0,0,0],[0,0,0,0],[9E9,9E9,9E9,9E9,9E9,9E9]];
    PERS bool P06W22_Used := FALSE;
    PERS num  P06W22_SubType := 0;
    PERS num  P06W22_ToolSel := 0;
    PERS num  P06W22_LenMM := 0;
    PERS robtarget P06W22_ArcStart := [[0,0,0],[1,0,0,0],[0,0,0,0],[9E9,9E9,9E9,9E9,9E9,9E9]];
    PERS robtarget P06W22_ArcEnd   := [[0,0,0],[1,0,0,0],[0,0,0,0],[9E9,9E9,9E9,9E9,9E9,9E9]];
    PERS robtarget P06W22_Approach := [[0,0,0],[1,0,0,0],[0,0,0,0],[9E9,9E9,9E9,9E9,9E9,9E9]];
    PERS robtarget P06W22_Retract  := [[0,0,0],[1,0,0,0],[0,0,0,0],[9E9,9E9,9E9,9E9,9E9,9E9]];
    PERS robtarget P06W22_Trans    := [[0,0,0],[1,0,0,0],[0,0,0,0],[9E9,9E9,9E9,9E9,9E9,9E9]];
    PERS bool P06W23_Used := FALSE;
    PERS num  P06W23_SubType := 0;
    PERS num  P06W23_ToolSel := 0;
    PERS num  P06W23_LenMM := 0;
    PERS robtarget P06W23_ArcStart := [[0,0,0],[1,0,0,0],[0,0,0,0],[9E9,9E9,9E9,9E9,9E9,9E9]];
    PERS robtarget P06W23_ArcEnd   := [[0,0,0],[1,0,0,0],[0,0,0,0],[9E9,9E9,9E9,9E9,9E9,9E9]];
    PERS robtarget P06W23_Approach := [[0,0,0],[1,0,0,0],[0,0,0,0],[9E9,9E9,9E9,9E9,9E9,9E9]];
    PERS robtarget P06W23_Retract  := [[0,0,0],[1,0,0,0],[0,0,0,0],[9E9,9E9,9E9,9E9,9E9,9E9]];
    PERS robtarget P06W23_Trans    := [[0,0,0],[1,0,0,0],[0,0,0,0],[9E9,9E9,9E9,9E9,9E9,9E9]];
    PERS bool P06W24_Used := FALSE;
    PERS num  P06W24_SubType := 0;
    PERS num  P06W24_ToolSel := 0;
    PERS num  P06W24_LenMM := 0;
    PERS robtarget P06W24_ArcStart := [[0,0,0],[1,0,0,0],[0,0,0,0],[9E9,9E9,9E9,9E9,9E9,9E9]];
    PERS robtarget P06W24_ArcEnd   := [[0,0,0],[1,0,0,0],[0,0,0,0],[9E9,9E9,9E9,9E9,9E9,9E9]];
    PERS robtarget P06W24_Approach := [[0,0,0],[1,0,0,0],[0,0,0,0],[9E9,9E9,9E9,9E9,9E9,9E9]];
    PERS robtarget P06W24_Retract  := [[0,0,0],[1,0,0,0],[0,0,0,0],[9E9,9E9,9E9,9E9,9E9,9E9]];
    PERS robtarget P06W24_Trans    := [[0,0,0],[1,0,0,0],[0,0,0,0],[9E9,9E9,9E9,9E9,9E9,9E9]];
    PERS bool P06W25_Used := FALSE;
    PERS num  P06W25_SubType := 0;
    PERS num  P06W25_ToolSel := 0;
    PERS num  P06W25_LenMM := 0;
    PERS robtarget P06W25_ArcStart := [[0,0,0],[1,0,0,0],[0,0,0,0],[9E9,9E9,9E9,9E9,9E9,9E9]];
    PERS robtarget P06W25_ArcEnd   := [[0,0,0],[1,0,0,0],[0,0,0,0],[9E9,9E9,9E9,9E9,9E9,9E9]];
    PERS robtarget P06W25_Approach := [[0,0,0],[1,0,0,0],[0,0,0,0],[9E9,9E9,9E9,9E9,9E9,9E9]];
    PERS robtarget P06W25_Retract  := [[0,0,0],[1,0,0,0],[0,0,0,0],[9E9,9E9,9E9,9E9,9E9,9E9]];
    PERS robtarget P06W25_Trans    := [[0,0,0],[1,0,0,0],[0,0,0,0],[9E9,9E9,9E9,9E9,9E9,9E9]];
    PERS bool P06W26_Used := FALSE;
    PERS num  P06W26_SubType := 0;
    PERS num  P06W26_ToolSel := 0;
    PERS num  P06W26_LenMM := 0;
    PERS robtarget P06W26_ArcStart := [[0,0,0],[1,0,0,0],[0,0,0,0],[9E9,9E9,9E9,9E9,9E9,9E9]];
    PERS robtarget P06W26_ArcEnd   := [[0,0,0],[1,0,0,0],[0,0,0,0],[9E9,9E9,9E9,9E9,9E9,9E9]];
    PERS robtarget P06W26_Approach := [[0,0,0],[1,0,0,0],[0,0,0,0],[9E9,9E9,9E9,9E9,9E9,9E9]];
    PERS robtarget P06W26_Retract  := [[0,0,0],[1,0,0,0],[0,0,0,0],[9E9,9E9,9E9,9E9,9E9,9E9]];
    PERS robtarget P06W26_Trans    := [[0,0,0],[1,0,0,0],[0,0,0,0],[9E9,9E9,9E9,9E9,9E9,9E9]];
    PERS bool P06W27_Used := FALSE;
    PERS num  P06W27_SubType := 0;
    PERS num  P06W27_ToolSel := 0;
    PERS num  P06W27_LenMM := 0;
    PERS robtarget P06W27_ArcStart := [[0,0,0],[1,0,0,0],[0,0,0,0],[9E9,9E9,9E9,9E9,9E9,9E9]];
    PERS robtarget P06W27_ArcEnd   := [[0,0,0],[1,0,0,0],[0,0,0,0],[9E9,9E9,9E9,9E9,9E9,9E9]];
    PERS robtarget P06W27_Approach := [[0,0,0],[1,0,0,0],[0,0,0,0],[9E9,9E9,9E9,9E9,9E9,9E9]];
    PERS robtarget P06W27_Retract  := [[0,0,0],[1,0,0,0],[0,0,0,0],[9E9,9E9,9E9,9E9,9E9,9E9]];
    PERS robtarget P06W27_Trans    := [[0,0,0],[1,0,0,0],[0,0,0,0],[9E9,9E9,9E9,9E9,9E9,9E9]];
    PERS bool P06W28_Used := FALSE;
    PERS num  P06W28_SubType := 0;
    PERS num  P06W28_ToolSel := 0;
    PERS num  P06W28_LenMM := 0;
    PERS robtarget P06W28_ArcStart := [[0,0,0],[1,0,0,0],[0,0,0,0],[9E9,9E9,9E9,9E9,9E9,9E9]];
    PERS robtarget P06W28_ArcEnd   := [[0,0,0],[1,0,0,0],[0,0,0,0],[9E9,9E9,9E9,9E9,9E9,9E9]];
    PERS robtarget P06W28_Approach := [[0,0,0],[1,0,0,0],[0,0,0,0],[9E9,9E9,9E9,9E9,9E9,9E9]];
    PERS robtarget P06W28_Retract  := [[0,0,0],[1,0,0,0],[0,0,0,0],[9E9,9E9,9E9,9E9,9E9,9E9]];
    PERS robtarget P06W28_Trans    := [[0,0,0],[1,0,0,0],[0,0,0,0],[9E9,9E9,9E9,9E9,9E9,9E9]];
    PERS bool P06W29_Used := FALSE;
    PERS num  P06W29_SubType := 0;
    PERS num  P06W29_ToolSel := 0;
    PERS num  P06W29_LenMM := 0;
    PERS robtarget P06W29_ArcStart := [[0,0,0],[1,0,0,0],[0,0,0,0],[9E9,9E9,9E9,9E9,9E9,9E9]];
    PERS robtarget P06W29_ArcEnd   := [[0,0,0],[1,0,0,0],[0,0,0,0],[9E9,9E9,9E9,9E9,9E9,9E9]];
    PERS robtarget P06W29_Approach := [[0,0,0],[1,0,0,0],[0,0,0,0],[9E9,9E9,9E9,9E9,9E9,9E9]];
    PERS robtarget P06W29_Retract  := [[0,0,0],[1,0,0,0],[0,0,0,0],[9E9,9E9,9E9,9E9,9E9,9E9]];
    PERS robtarget P06W29_Trans    := [[0,0,0],[1,0,0,0],[0,0,0,0],[9E9,9E9,9E9,9E9,9E9,9E9]];
    PERS bool P06W30_Used := FALSE;
    PERS num  P06W30_SubType := 0;
    PERS num  P06W30_ToolSel := 0;
    PERS num  P06W30_LenMM := 0;
    PERS robtarget P06W30_ArcStart := [[0,0,0],[1,0,0,0],[0,0,0,0],[9E9,9E9,9E9,9E9,9E9,9E9]];
    PERS robtarget P06W30_ArcEnd   := [[0,0,0],[1,0,0,0],[0,0,0,0],[9E9,9E9,9E9,9E9,9E9,9E9]];
    PERS robtarget P06W30_Approach := [[0,0,0],[1,0,0,0],[0,0,0,0],[9E9,9E9,9E9,9E9,9E9,9E9]];
    PERS robtarget P06W30_Retract  := [[0,0,0],[1,0,0,0],[0,0,0,0],[9E9,9E9,9E9,9E9,9E9,9E9]];
    PERS robtarget P06W30_Trans    := [[0,0,0],[1,0,0,0],[0,0,0,0],[9E9,9E9,9E9,9E9,9E9,9E9]];

    ! =========================
    ! ======= CONSTANTS =======
    ! =========================
    CONST num INCH := 25.4;
    CONST num cApproach := 0.100*INCH;
    CONST num cTransZ   := 10.0*INCH;

    CONST num WT_VERT   := 1;
    CONST num WT_HORIZ  := 2;
    CONST num WT_CORNER := 3;
    CONST num WT_FREE   := 4;

    CONST num WSV_YLEFT  := 11;
    CONST num WSV_YRIGHT := 12;
    CONST num WSV_YMID   := 13;
    CONST num WSH_XUP    := 21;
    CONST num WSH_XDN    := 22;
    CONST num WSH_XMID   := 23;
    CONST num WSC_ULC    := 31;
    CONST num WSC_URC    := 32;
    CONST num WSC_DLC    := 33;
    CONST num WSC_DRC    := 34;
    CONST num WSF_FREE   := 41;

    CONST num T_OLEFT := 1;
    CONST num T_ORIGHT:= 2;
    CONST num T_OUP   := 3;
    CONST num T_ODOWN := 4;
    CONST num T_OYMID := 5;
    CONST num T_OXMID := 6;

    PROC LoadDefaultWeldData(VAR seamdata seamOut, VAR welddata weldOut, VAR weavedata weaveOut)
        seamOut := cSeamDefault;
        weldOut := cWeldDefault;
        weaveOut := cWeaveDefault;
    ENDPROC

    ! =========================
    ! ===== ORI PICKER ========
    ! =========================
    FUNC robtarget GetOriPose(num toolSel)
        IF toolSel = T_OLEFT THEN
            RETURN pOri_Left;
        ELSEIF toolSel = T_ORIGHT THEN
            RETURN pOri_Right;
        ELSEIF toolSel = T_OUP THEN
            RETURN pOri_Up;
        ELSEIF toolSel = T_ODOWN THEN
            RETURN pOri_Down;
        ELSEIF toolSel = T_OYMID THEN
            RETURN pOri_yMid;
        ELSE
            RETURN pOri_xMid;
        ENDIF
    ENDFUNC

    ! =========================
    ! ===== GEOMETRY ==========
    ! =========================
    FUNC robtarget CalcApproach(robtarget arcStart, num subType)
        IF subType = WSV_YLEFT THEN
            RETURN Offs(arcStart, -cApproach, +cApproach, +cApproach);
        ELSEIF subType = WSV_YRIGHT THEN
            RETURN Offs(arcStart, +cApproach, +cApproach, +cApproach);
        ELSEIF subType = WSH_XUP THEN
            RETURN Offs(arcStart, -cApproach, +cApproach, +cApproach);
        ELSEIF subType = WSH_XDN THEN
            RETURN Offs(arcStart, -cApproach, -cApproach, +cApproach);
        ELSE
            RETURN Offs(arcStart, 0, 0, +cApproach);
        ENDIF
    ENDFUNC

    FUNC robtarget CalcArcEnd(robtarget arcStart, num subType, num lenMM, robtarget freeEnd)
        IF subType = WSV_YLEFT OR subType = WSV_YRIGHT OR subType = WSV_YMID THEN
            RETURN Offs(arcStart, 0, -lenMM, 0);
        ELSEIF subType = WSH_XUP OR subType = WSH_XDN OR subType = WSH_XMID THEN
            RETURN Offs(arcStart, +lenMM, 0, 0);
        ELSE
            RETURN freeEnd;
        ENDIF
    ENDFUNC

    FUNC robtarget CalcRetract(robtarget arcEnd, num subType)
        IF subType = WSV_YLEFT THEN
            RETURN Offs(arcEnd, -cApproach, +cApproach, +cApproach);
        ELSEIF subType = WSV_YRIGHT THEN
            RETURN Offs(arcEnd, +cApproach, +cApproach, +cApproach);
        ELSEIF subType = WSH_XUP THEN
            RETURN Offs(arcEnd, -cApproach, +cApproach, +cApproach);
        ELSEIF subType = WSH_XDN THEN
            RETURN Offs(arcEnd, -cApproach, -cApproach, +cApproach);
        ELSE
            RETURN Offs(arcEnd, 0, 0, +cApproach);
        ENDIF
    ENDFUNC

    FUNC robtarget CalcTransverse(robtarget retract)
        RETURN Offs(retract, 0, 0, +cTransZ);
    ENDFUNC

    FUNC robtarget ApplyOri(robtarget p, num toolSel)
        VAR robtarget o;
        o := GetOriPose(toolSel);
        p.rot := o.rot;
        p.robconf := o.robconf;
        p.extax := o.extax;
        RETURN p;
    ENDFUNC

    PROC MoveToTeachOrientation(num toolSel)
        VAR robtarget pOriSafe;
        MoveJ pSafeS1Weld, v200, z50, tWeldGun;
        pOriSafe := ApplyOri(pSafeS1Weld, toolSel);
        MoveJ pOriSafe, v200, z50, tWeldGun;
    ENDPROC

    PROC BuildWeldFromStart(
        robtarget startIn,
        robtarget freeEndIn,
        num subType,
        num toolSel,
        num lenMM,
        VAR robtarget arcStart,
        VAR robtarget arcEnd,
        VAR robtarget approach,
        VAR robtarget retract,
        VAR robtarget trans)
        arcStart := startIn;
        arcStart := ApplyOri(arcStart, toolSel);
        arcEnd := CalcArcEnd(arcStart, subType, lenMM, freeEndIn);
        arcEnd := ApplyOri(arcEnd, toolSel);
        approach := CalcApproach(arcStart, subType);
        approach := ApplyOri(approach, toolSel);
        retract := CalcRetract(arcEnd, subType);
        retract := ApplyOri(retract, toolSel);
        trans := CalcTransverse(retract);
        trans := ApplyOri(trans, toolSel);
    ENDPROC

    ! =========================
    ! ==== DRY RUN MOVE =======
    ! =========================
    PROC DryRun(robtarget pTrans, robtarget pApp, robtarget pS, robtarget pE, robtarget pRet)
        MoveL pTrans, vPreviewTrans, z50, tWeldGun;
        MoveL pApp,   vPreviewApproach, z10, tWeldGun;
        MoveL pS,     vPreviewArcStart, z1,  tWeldGun;
        MoveL pE,     vPreviewArcEnd, z1,  tWeldGun;
        MoveL pRet,   vPreviewRetract, z10, tWeldGun;
        MoveL pTrans, vPreviewTrans, z50, tWeldGun;
    ENDPROC

    PROC SetupP01()
        MoveJ pSetup, v200, z50, tWeldGun;
        TPWrite "Jog to Origin 1 Base (most x-,y-). Press Play.";
        Stop \NoRegain;
        P01Origin := CRobT(\Tool:=tWeldGun);
        TPWrite "Jog to Origin 1 Limit (most x+,y+). Press Play.";
        Stop \NoRegain;
        P01Max := CRobT(\Tool:=tWeldGun);
        TPWrite "Jog to Origin 1 Z-Plane (touch wire tip). Press Play.";
        Stop \NoRegain;
        P01Zoff := CRobT(\Tool:=tWeldGun);
        wobjP01.uframe.trans := P01Origin.trans;
        wobjP01.uframe.rot := P01Origin.rot;
        wobjP01.oframe.trans := P01Zoff.trans;
        wobjP01.oframe.rot := P01Zoff.rot;
        TPWrite "Origin 1 points recorded.";
        MoveJ pSafeS1Weld, v200, z50, tWeldGun;
    ENDPROC

    PROC SetupP02()
        MoveJ pSetup, v200, z50, tWeldGun;
        TPWrite "Jog to Origin 2 Base (most x-,y-). Press Play.";
        Stop \NoRegain;
        P02Origin := CRobT(\Tool:=tWeldGun);
        TPWrite "Jog to Origin 2 Limit (most x+,y+). Press Play.";
        Stop \NoRegain;
        P02Max := CRobT(\Tool:=tWeldGun);
        TPWrite "Jog to Origin 2 Z-Plane (touch wire tip). Press Play.";
        Stop \NoRegain;
        P02Zoff := CRobT(\Tool:=tWeldGun);
        wobjP02.uframe.trans := P02Origin.trans;
        wobjP02.uframe.rot := P02Origin.rot;
        wobjP02.oframe.trans := P02Zoff.trans;
        wobjP02.oframe.rot := P02Zoff.rot;
        TPWrite "Origin 2 points recorded.";
        MoveJ pSafeS1Weld, v200, z50, tWeldGun;
    ENDPROC

    PROC SetupP03()
        MoveJ pSetup, v200, z50, tWeldGun;
        TPWrite "Jog to Origin 3 Base (most x-,y-). Press Play.";
        Stop \NoRegain;
        P03Origin := CRobT(\Tool:=tWeldGun);
        TPWrite "Jog to Origin 3 Limit (most x+,y+). Press Play.";
        Stop \NoRegain;
        P03Max := CRobT(\Tool:=tWeldGun);
        TPWrite "Jog to Origin 3 Z-Plane (touch wire tip). Press Play.";
        Stop \NoRegain;
        P03Zoff := CRobT(\Tool:=tWeldGun);
        wobjP03.uframe.trans := P03Origin.trans;
        wobjP03.uframe.rot := P03Origin.rot;
        wobjP03.oframe.trans := P03Zoff.trans;
        wobjP03.oframe.rot := P03Zoff.rot;
        TPWrite "Origin 3 points recorded.";
        MoveJ pSafeS1Weld, v200, z50, tWeldGun;
    ENDPROC

    PROC SetupP04()
        MoveJ pSetup, v200, z50, tWeldGun;
        TPWrite "Jog to Origin 4 Base (most x-,y-). Press Play.";
        Stop \NoRegain;
        P04Origin := CRobT(\Tool:=tWeldGun);
        TPWrite "Jog to Origin 4 Limit (most x+,y+). Press Play.";
        Stop \NoRegain;
        P04Max := CRobT(\Tool:=tWeldGun);
        TPWrite "Jog to Origin 4 Z-Plane (touch wire tip). Press Play.";
        Stop \NoRegain;
        P04Zoff := CRobT(\Tool:=tWeldGun);
        wobjP04.uframe.trans := P04Origin.trans;
        wobjP04.uframe.rot := P04Origin.rot;
        wobjP04.oframe.trans := P04Zoff.trans;
        wobjP04.oframe.rot := P04Zoff.rot;
        TPWrite "Origin 4 points recorded.";
        MoveJ pSafeS1Weld, v200, z50, tWeldGun;
    ENDPROC

    PROC SetupP05()
        MoveJ pSetup, v200, z50, tWeldGun;
        TPWrite "Jog to Origin 5 Base (most x-,y-). Press Play.";
        Stop \NoRegain;
        P05Origin := CRobT(\Tool:=tWeldGun);
        TPWrite "Jog to Origin 5 Limit (most x+,y+). Press Play.";
        Stop \NoRegain;
        P05Max := CRobT(\Tool:=tWeldGun);
        TPWrite "Jog to Origin 5 Z-Plane (touch wire tip). Press Play.";
        Stop \NoRegain;
        P05Zoff := CRobT(\Tool:=tWeldGun);
        wobjP05.uframe.trans := P05Origin.trans;
        wobjP05.uframe.rot := P05Origin.rot;
        wobjP05.oframe.trans := P05Zoff.trans;
        wobjP05.oframe.rot := P05Zoff.rot;
        TPWrite "Origin 5 points recorded.";
        MoveJ pSafeS1Weld, v200, z50, tWeldGun;
    ENDPROC

    PROC SetupP06()
        MoveJ pSetup, v200, z50, tWeldGun;
        TPWrite "Jog to Origin 6 Base (most x-,y-). Press Play.";
        Stop \NoRegain;
        P06Origin := CRobT(\Tool:=tWeldGun);
        TPWrite "Jog to Origin 6 Limit (most x+,y+). Press Play.";
        Stop \NoRegain;
        P06Max := CRobT(\Tool:=tWeldGun);
        TPWrite "Jog to Origin 6 Z-Plane (touch wire tip). Press Play.";
        Stop \NoRegain;
        P06Zoff := CRobT(\Tool:=tWeldGun);
        wobjP06.uframe.trans := P06Origin.trans;
        wobjP06.uframe.rot := P06Origin.rot;
        wobjP06.oframe.trans := P06Zoff.trans;
        wobjP06.oframe.rot := P06Zoff.rot;
        TPWrite "Origin 6 points recorded.";
        MoveJ pSafeS1Weld, v200, z50, tWeldGun;
    ENDPROC

    PROC TeachOrientation(num toolSel)
        MoveJ pSafeS1, v200, z50, tWeldGun;
        TPWrite "Jog from pSafeS1 down to bullseye/orientation, then press Play.";
        Stop \NoRegain;
        IF toolSel = T_OLEFT THEN
            pOri_Left := CRobT(\Tool:=tWeldGun);
        ELSEIF toolSel = T_ORIGHT THEN
            pOri_Right := CRobT(\Tool:=tWeldGun);
        ELSEIF toolSel = T_OUP THEN
            pOri_Up := CRobT(\Tool:=tWeldGun);
        ELSEIF toolSel = T_ODOWN THEN
            pOri_Down := CRobT(\Tool:=tWeldGun);
        ELSEIF toolSel = T_OYMID THEN
            pOri_yMid := CRobT(\Tool:=tWeldGun);
        ELSE
            pOri_xMid := CRobT(\Tool:=tWeldGun);
        ENDIF
        TPWrite "Orientation stored.";
        MoveJ pSafeS1, v200, z50, tWeldGun;
    ENDPROC

    PROC StoreSlot_P01(num slot, num subType, num toolSel, num lenMM,
                       robtarget arcStart, robtarget arcEnd, robtarget approach, robtarget retract, robtarget trans)
        IF slot = 1 THEN
            P01W01_SubType := subType;
            P01W01_ToolSel := toolSel;
            P01W01_LenMM := lenMM;
            P01W01_ArcStart := arcStart;
            P01W01_ArcEnd := arcEnd;
            P01W01_Approach := approach;
            P01W01_Retract := retract;
            P01W01_Trans := trans;
            P01W01_Used := TRUE;
        ELSEIF slot = 2 THEN
            P01W02_SubType := subType;
            P01W02_ToolSel := toolSel;
            P01W02_LenMM := lenMM;
            P01W02_ArcStart := arcStart;
            P01W02_ArcEnd := arcEnd;
            P01W02_Approach := approach;
            P01W02_Retract := retract;
            P01W02_Trans := trans;
            P01W02_Used := TRUE;
        ELSEIF slot = 3 THEN
            P01W03_SubType := subType;
            P01W03_ToolSel := toolSel;
            P01W03_LenMM := lenMM;
            P01W03_ArcStart := arcStart;
            P01W03_ArcEnd := arcEnd;
            P01W03_Approach := approach;
            P01W03_Retract := retract;
            P01W03_Trans := trans;
            P01W03_Used := TRUE;
        ELSEIF slot = 4 THEN
            P01W04_SubType := subType;
            P01W04_ToolSel := toolSel;
            P01W04_LenMM := lenMM;
            P01W04_ArcStart := arcStart;
            P01W04_ArcEnd := arcEnd;
            P01W04_Approach := approach;
            P01W04_Retract := retract;
            P01W04_Trans := trans;
            P01W04_Used := TRUE;
        ELSEIF slot = 5 THEN
            P01W05_SubType := subType;
            P01W05_ToolSel := toolSel;
            P01W05_LenMM := lenMM;
            P01W05_ArcStart := arcStart;
            P01W05_ArcEnd := arcEnd;
            P01W05_Approach := approach;
            P01W05_Retract := retract;
            P01W05_Trans := trans;
            P01W05_Used := TRUE;
        ELSEIF slot = 6 THEN
            P01W06_SubType := subType;
            P01W06_ToolSel := toolSel;
            P01W06_LenMM := lenMM;
            P01W06_ArcStart := arcStart;
            P01W06_ArcEnd := arcEnd;
            P01W06_Approach := approach;
            P01W06_Retract := retract;
            P01W06_Trans := trans;
            P01W06_Used := TRUE;
        ELSEIF slot = 7 THEN
            P01W07_SubType := subType;
            P01W07_ToolSel := toolSel;
            P01W07_LenMM := lenMM;
            P01W07_ArcStart := arcStart;
            P01W07_ArcEnd := arcEnd;
            P01W07_Approach := approach;
            P01W07_Retract := retract;
            P01W07_Trans := trans;
            P01W07_Used := TRUE;
        ELSEIF slot = 8 THEN
            P01W08_SubType := subType;
            P01W08_ToolSel := toolSel;
            P01W08_LenMM := lenMM;
            P01W08_ArcStart := arcStart;
            P01W08_ArcEnd := arcEnd;
            P01W08_Approach := approach;
            P01W08_Retract := retract;
            P01W08_Trans := trans;
            P01W08_Used := TRUE;
        ELSEIF slot = 9 THEN
            P01W09_SubType := subType;
            P01W09_ToolSel := toolSel;
            P01W09_LenMM := lenMM;
            P01W09_ArcStart := arcStart;
            P01W09_ArcEnd := arcEnd;
            P01W09_Approach := approach;
            P01W09_Retract := retract;
            P01W09_Trans := trans;
            P01W09_Used := TRUE;
        ELSEIF slot = 10 THEN
            P01W10_SubType := subType;
            P01W10_ToolSel := toolSel;
            P01W10_LenMM := lenMM;
            P01W10_ArcStart := arcStart;
            P01W10_ArcEnd := arcEnd;
            P01W10_Approach := approach;
            P01W10_Retract := retract;
            P01W10_Trans := trans;
            P01W10_Used := TRUE;
        ELSEIF slot = 11 THEN
            P01W11_SubType := subType;
            P01W11_ToolSel := toolSel;
            P01W11_LenMM := lenMM;
            P01W11_ArcStart := arcStart;
            P01W11_ArcEnd := arcEnd;
            P01W11_Approach := approach;
            P01W11_Retract := retract;
            P01W11_Trans := trans;
            P01W11_Used := TRUE;
        ELSEIF slot = 12 THEN
            P01W12_SubType := subType;
            P01W12_ToolSel := toolSel;
            P01W12_LenMM := lenMM;
            P01W12_ArcStart := arcStart;
            P01W12_ArcEnd := arcEnd;
            P01W12_Approach := approach;
            P01W12_Retract := retract;
            P01W12_Trans := trans;
            P01W12_Used := TRUE;
        ELSEIF slot = 13 THEN
            P01W13_SubType := subType;
            P01W13_ToolSel := toolSel;
            P01W13_LenMM := lenMM;
            P01W13_ArcStart := arcStart;
            P01W13_ArcEnd := arcEnd;
            P01W13_Approach := approach;
            P01W13_Retract := retract;
            P01W13_Trans := trans;
            P01W13_Used := TRUE;
        ELSEIF slot = 14 THEN
            P01W14_SubType := subType;
            P01W14_ToolSel := toolSel;
            P01W14_LenMM := lenMM;
            P01W14_ArcStart := arcStart;
            P01W14_ArcEnd := arcEnd;
            P01W14_Approach := approach;
            P01W14_Retract := retract;
            P01W14_Trans := trans;
            P01W14_Used := TRUE;
        ELSEIF slot = 15 THEN
            P01W15_SubType := subType;
            P01W15_ToolSel := toolSel;
            P01W15_LenMM := lenMM;
            P01W15_ArcStart := arcStart;
            P01W15_ArcEnd := arcEnd;
            P01W15_Approach := approach;
            P01W15_Retract := retract;
            P01W15_Trans := trans;
            P01W15_Used := TRUE;
        ELSEIF slot = 16 THEN
            P01W16_SubType := subType;
            P01W16_ToolSel := toolSel;
            P01W16_LenMM := lenMM;
            P01W16_ArcStart := arcStart;
            P01W16_ArcEnd := arcEnd;
            P01W16_Approach := approach;
            P01W16_Retract := retract;
            P01W16_Trans := trans;
            P01W16_Used := TRUE;
        ELSEIF slot = 17 THEN
            P01W17_SubType := subType;
            P01W17_ToolSel := toolSel;
            P01W17_LenMM := lenMM;
            P01W17_ArcStart := arcStart;
            P01W17_ArcEnd := arcEnd;
            P01W17_Approach := approach;
            P01W17_Retract := retract;
            P01W17_Trans := trans;
            P01W17_Used := TRUE;
        ELSEIF slot = 18 THEN
            P01W18_SubType := subType;
            P01W18_ToolSel := toolSel;
            P01W18_LenMM := lenMM;
            P01W18_ArcStart := arcStart;
            P01W18_ArcEnd := arcEnd;
            P01W18_Approach := approach;
            P01W18_Retract := retract;
            P01W18_Trans := trans;
            P01W18_Used := TRUE;
        ELSEIF slot = 19 THEN
            P01W19_SubType := subType;
            P01W19_ToolSel := toolSel;
            P01W19_LenMM := lenMM;
            P01W19_ArcStart := arcStart;
            P01W19_ArcEnd := arcEnd;
            P01W19_Approach := approach;
            P01W19_Retract := retract;
            P01W19_Trans := trans;
            P01W19_Used := TRUE;
        ELSEIF slot = 20 THEN
            P01W20_SubType := subType;
            P01W20_ToolSel := toolSel;
            P01W20_LenMM := lenMM;
            P01W20_ArcStart := arcStart;
            P01W20_ArcEnd := arcEnd;
            P01W20_Approach := approach;
            P01W20_Retract := retract;
            P01W20_Trans := trans;
            P01W20_Used := TRUE;
        ELSEIF slot = 21 THEN
            P01W21_SubType := subType;
            P01W21_ToolSel := toolSel;
            P01W21_LenMM := lenMM;
            P01W21_ArcStart := arcStart;
            P01W21_ArcEnd := arcEnd;
            P01W21_Approach := approach;
            P01W21_Retract := retract;
            P01W21_Trans := trans;
            P01W21_Used := TRUE;
        ELSEIF slot = 22 THEN
            P01W22_SubType := subType;
            P01W22_ToolSel := toolSel;
            P01W22_LenMM := lenMM;
            P01W22_ArcStart := arcStart;
            P01W22_ArcEnd := arcEnd;
            P01W22_Approach := approach;
            P01W22_Retract := retract;
            P01W22_Trans := trans;
            P01W22_Used := TRUE;
        ELSEIF slot = 23 THEN
            P01W23_SubType := subType;
            P01W23_ToolSel := toolSel;
            P01W23_LenMM := lenMM;
            P01W23_ArcStart := arcStart;
            P01W23_ArcEnd := arcEnd;
            P01W23_Approach := approach;
            P01W23_Retract := retract;
            P01W23_Trans := trans;
            P01W23_Used := TRUE;
        ELSEIF slot = 24 THEN
            P01W24_SubType := subType;
            P01W24_ToolSel := toolSel;
            P01W24_LenMM := lenMM;
            P01W24_ArcStart := arcStart;
            P01W24_ArcEnd := arcEnd;
            P01W24_Approach := approach;
            P01W24_Retract := retract;
            P01W24_Trans := trans;
            P01W24_Used := TRUE;
        ELSEIF slot = 25 THEN
            P01W25_SubType := subType;
            P01W25_ToolSel := toolSel;
            P01W25_LenMM := lenMM;
            P01W25_ArcStart := arcStart;
            P01W25_ArcEnd := arcEnd;
            P01W25_Approach := approach;
            P01W25_Retract := retract;
            P01W25_Trans := trans;
            P01W25_Used := TRUE;
        ELSEIF slot = 26 THEN
            P01W26_SubType := subType;
            P01W26_ToolSel := toolSel;
            P01W26_LenMM := lenMM;
            P01W26_ArcStart := arcStart;
            P01W26_ArcEnd := arcEnd;
            P01W26_Approach := approach;
            P01W26_Retract := retract;
            P01W26_Trans := trans;
            P01W26_Used := TRUE;
        ELSEIF slot = 27 THEN
            P01W27_SubType := subType;
            P01W27_ToolSel := toolSel;
            P01W27_LenMM := lenMM;
            P01W27_ArcStart := arcStart;
            P01W27_ArcEnd := arcEnd;
            P01W27_Approach := approach;
            P01W27_Retract := retract;
            P01W27_Trans := trans;
            P01W27_Used := TRUE;
        ELSEIF slot = 28 THEN
            P01W28_SubType := subType;
            P01W28_ToolSel := toolSel;
            P01W28_LenMM := lenMM;
            P01W28_ArcStart := arcStart;
            P01W28_ArcEnd := arcEnd;
            P01W28_Approach := approach;
            P01W28_Retract := retract;
            P01W28_Trans := trans;
            P01W28_Used := TRUE;
        ELSEIF slot = 29 THEN
            P01W29_SubType := subType;
            P01W29_ToolSel := toolSel;
            P01W29_LenMM := lenMM;
            P01W29_ArcStart := arcStart;
            P01W29_ArcEnd := arcEnd;
            P01W29_Approach := approach;
            P01W29_Retract := retract;
            P01W29_Trans := trans;
            P01W29_Used := TRUE;
        ELSEIF slot = 30 THEN
            P01W30_SubType := subType;
            P01W30_ToolSel := toolSel;
            P01W30_LenMM := lenMM;
            P01W30_ArcStart := arcStart;
            P01W30_ArcEnd := arcEnd;
            P01W30_Approach := approach;
            P01W30_Retract := retract;
            P01W30_Trans := trans;
            P01W30_Used := TRUE;
        ELSE
            TPWrite "Invalid weld slot.";
        ENDIF
    ENDPROC

    PROC LoadSlot_P01(num slot, VAR bool used, VAR num subType, VAR num toolSel, VAR num lenMM,
                       VAR robtarget arcStart, VAR robtarget arcEnd, VAR robtarget approach, VAR robtarget retract, VAR robtarget trans)
        IF slot = 1 THEN
            used := P01W01_Used;
            subType := P01W01_SubType;
            toolSel := P01W01_ToolSel;
            lenMM := P01W01_LenMM;
            arcStart := P01W01_ArcStart;
            arcEnd := P01W01_ArcEnd;
            approach := P01W01_Approach;
            retract := P01W01_Retract;
            trans := P01W01_Trans;
        ELSEIF slot = 2 THEN
            used := P01W02_Used;
            subType := P01W02_SubType;
            toolSel := P01W02_ToolSel;
            lenMM := P01W02_LenMM;
            arcStart := P01W02_ArcStart;
            arcEnd := P01W02_ArcEnd;
            approach := P01W02_Approach;
            retract := P01W02_Retract;
            trans := P01W02_Trans;
        ELSEIF slot = 3 THEN
            used := P01W03_Used;
            subType := P01W03_SubType;
            toolSel := P01W03_ToolSel;
            lenMM := P01W03_LenMM;
            arcStart := P01W03_ArcStart;
            arcEnd := P01W03_ArcEnd;
            approach := P01W03_Approach;
            retract := P01W03_Retract;
            trans := P01W03_Trans;
        ELSEIF slot = 4 THEN
            used := P01W04_Used;
            subType := P01W04_SubType;
            toolSel := P01W04_ToolSel;
            lenMM := P01W04_LenMM;
            arcStart := P01W04_ArcStart;
            arcEnd := P01W04_ArcEnd;
            approach := P01W04_Approach;
            retract := P01W04_Retract;
            trans := P01W04_Trans;
        ELSEIF slot = 5 THEN
            used := P01W05_Used;
            subType := P01W05_SubType;
            toolSel := P01W05_ToolSel;
            lenMM := P01W05_LenMM;
            arcStart := P01W05_ArcStart;
            arcEnd := P01W05_ArcEnd;
            approach := P01W05_Approach;
            retract := P01W05_Retract;
            trans := P01W05_Trans;
        ELSEIF slot = 6 THEN
            used := P01W06_Used;
            subType := P01W06_SubType;
            toolSel := P01W06_ToolSel;
            lenMM := P01W06_LenMM;
            arcStart := P01W06_ArcStart;
            arcEnd := P01W06_ArcEnd;
            approach := P01W06_Approach;
            retract := P01W06_Retract;
            trans := P01W06_Trans;
        ELSEIF slot = 7 THEN
            used := P01W07_Used;
            subType := P01W07_SubType;
            toolSel := P01W07_ToolSel;
            lenMM := P01W07_LenMM;
            arcStart := P01W07_ArcStart;
            arcEnd := P01W07_ArcEnd;
            approach := P01W07_Approach;
            retract := P01W07_Retract;
            trans := P01W07_Trans;
        ELSEIF slot = 8 THEN
            used := P01W08_Used;
            subType := P01W08_SubType;
            toolSel := P01W08_ToolSel;
            lenMM := P01W08_LenMM;
            arcStart := P01W08_ArcStart;
            arcEnd := P01W08_ArcEnd;
            approach := P01W08_Approach;
            retract := P01W08_Retract;
            trans := P01W08_Trans;
        ELSEIF slot = 9 THEN
            used := P01W09_Used;
            subType := P01W09_SubType;
            toolSel := P01W09_ToolSel;
            lenMM := P01W09_LenMM;
            arcStart := P01W09_ArcStart;
            arcEnd := P01W09_ArcEnd;
            approach := P01W09_Approach;
            retract := P01W09_Retract;
            trans := P01W09_Trans;
        ELSEIF slot = 10 THEN
            used := P01W10_Used;
            subType := P01W10_SubType;
            toolSel := P01W10_ToolSel;
            lenMM := P01W10_LenMM;
            arcStart := P01W10_ArcStart;
            arcEnd := P01W10_ArcEnd;
            approach := P01W10_Approach;
            retract := P01W10_Retract;
            trans := P01W10_Trans;
        ELSEIF slot = 11 THEN
            used := P01W11_Used;
            subType := P01W11_SubType;
            toolSel := P01W11_ToolSel;
            lenMM := P01W11_LenMM;
            arcStart := P01W11_ArcStart;
            arcEnd := P01W11_ArcEnd;
            approach := P01W11_Approach;
            retract := P01W11_Retract;
            trans := P01W11_Trans;
        ELSEIF slot = 12 THEN
            used := P01W12_Used;
            subType := P01W12_SubType;
            toolSel := P01W12_ToolSel;
            lenMM := P01W12_LenMM;
            arcStart := P01W12_ArcStart;
            arcEnd := P01W12_ArcEnd;
            approach := P01W12_Approach;
            retract := P01W12_Retract;
            trans := P01W12_Trans;
        ELSEIF slot = 13 THEN
            used := P01W13_Used;
            subType := P01W13_SubType;
            toolSel := P01W13_ToolSel;
            lenMM := P01W13_LenMM;
            arcStart := P01W13_ArcStart;
            arcEnd := P01W13_ArcEnd;
            approach := P01W13_Approach;
            retract := P01W13_Retract;
            trans := P01W13_Trans;
        ELSEIF slot = 14 THEN
            used := P01W14_Used;
            subType := P01W14_SubType;
            toolSel := P01W14_ToolSel;
            lenMM := P01W14_LenMM;
            arcStart := P01W14_ArcStart;
            arcEnd := P01W14_ArcEnd;
            approach := P01W14_Approach;
            retract := P01W14_Retract;
            trans := P01W14_Trans;
        ELSEIF slot = 15 THEN
            used := P01W15_Used;
            subType := P01W15_SubType;
            toolSel := P01W15_ToolSel;
            lenMM := P01W15_LenMM;
            arcStart := P01W15_ArcStart;
            arcEnd := P01W15_ArcEnd;
            approach := P01W15_Approach;
            retract := P01W15_Retract;
            trans := P01W15_Trans;
        ELSEIF slot = 16 THEN
            used := P01W16_Used;
            subType := P01W16_SubType;
            toolSel := P01W16_ToolSel;
            lenMM := P01W16_LenMM;
            arcStart := P01W16_ArcStart;
            arcEnd := P01W16_ArcEnd;
            approach := P01W16_Approach;
            retract := P01W16_Retract;
            trans := P01W16_Trans;
        ELSEIF slot = 17 THEN
            used := P01W17_Used;
            subType := P01W17_SubType;
            toolSel := P01W17_ToolSel;
            lenMM := P01W17_LenMM;
            arcStart := P01W17_ArcStart;
            arcEnd := P01W17_ArcEnd;
            approach := P01W17_Approach;
            retract := P01W17_Retract;
            trans := P01W17_Trans;
        ELSEIF slot = 18 THEN
            used := P01W18_Used;
            subType := P01W18_SubType;
            toolSel := P01W18_ToolSel;
            lenMM := P01W18_LenMM;
            arcStart := P01W18_ArcStart;
            arcEnd := P01W18_ArcEnd;
            approach := P01W18_Approach;
            retract := P01W18_Retract;
            trans := P01W18_Trans;
        ELSEIF slot = 19 THEN
            used := P01W19_Used;
            subType := P01W19_SubType;
            toolSel := P01W19_ToolSel;
            lenMM := P01W19_LenMM;
            arcStart := P01W19_ArcStart;
            arcEnd := P01W19_ArcEnd;
            approach := P01W19_Approach;
            retract := P01W19_Retract;
            trans := P01W19_Trans;
        ELSEIF slot = 20 THEN
            used := P01W20_Used;
            subType := P01W20_SubType;
            toolSel := P01W20_ToolSel;
            lenMM := P01W20_LenMM;
            arcStart := P01W20_ArcStart;
            arcEnd := P01W20_ArcEnd;
            approach := P01W20_Approach;
            retract := P01W20_Retract;
            trans := P01W20_Trans;
        ELSEIF slot = 21 THEN
            used := P01W21_Used;
            subType := P01W21_SubType;
            toolSel := P01W21_ToolSel;
            lenMM := P01W21_LenMM;
            arcStart := P01W21_ArcStart;
            arcEnd := P01W21_ArcEnd;
            approach := P01W21_Approach;
            retract := P01W21_Retract;
            trans := P01W21_Trans;
        ELSEIF slot = 22 THEN
            used := P01W22_Used;
            subType := P01W22_SubType;
            toolSel := P01W22_ToolSel;
            lenMM := P01W22_LenMM;
            arcStart := P01W22_ArcStart;
            arcEnd := P01W22_ArcEnd;
            approach := P01W22_Approach;
            retract := P01W22_Retract;
            trans := P01W22_Trans;
        ELSEIF slot = 23 THEN
            used := P01W23_Used;
            subType := P01W23_SubType;
            toolSel := P01W23_ToolSel;
            lenMM := P01W23_LenMM;
            arcStart := P01W23_ArcStart;
            arcEnd := P01W23_ArcEnd;
            approach := P01W23_Approach;
            retract := P01W23_Retract;
            trans := P01W23_Trans;
        ELSEIF slot = 24 THEN
            used := P01W24_Used;
            subType := P01W24_SubType;
            toolSel := P01W24_ToolSel;
            lenMM := P01W24_LenMM;
            arcStart := P01W24_ArcStart;
            arcEnd := P01W24_ArcEnd;
            approach := P01W24_Approach;
            retract := P01W24_Retract;
            trans := P01W24_Trans;
        ELSEIF slot = 25 THEN
            used := P01W25_Used;
            subType := P01W25_SubType;
            toolSel := P01W25_ToolSel;
            lenMM := P01W25_LenMM;
            arcStart := P01W25_ArcStart;
            arcEnd := P01W25_ArcEnd;
            approach := P01W25_Approach;
            retract := P01W25_Retract;
            trans := P01W25_Trans;
        ELSEIF slot = 26 THEN
            used := P01W26_Used;
            subType := P01W26_SubType;
            toolSel := P01W26_ToolSel;
            lenMM := P01W26_LenMM;
            arcStart := P01W26_ArcStart;
            arcEnd := P01W26_ArcEnd;
            approach := P01W26_Approach;
            retract := P01W26_Retract;
            trans := P01W26_Trans;
        ELSEIF slot = 27 THEN
            used := P01W27_Used;
            subType := P01W27_SubType;
            toolSel := P01W27_ToolSel;
            lenMM := P01W27_LenMM;
            arcStart := P01W27_ArcStart;
            arcEnd := P01W27_ArcEnd;
            approach := P01W27_Approach;
            retract := P01W27_Retract;
            trans := P01W27_Trans;
        ELSEIF slot = 28 THEN
            used := P01W28_Used;
            subType := P01W28_SubType;
            toolSel := P01W28_ToolSel;
            lenMM := P01W28_LenMM;
            arcStart := P01W28_ArcStart;
            arcEnd := P01W28_ArcEnd;
            approach := P01W28_Approach;
            retract := P01W28_Retract;
            trans := P01W28_Trans;
        ELSEIF slot = 29 THEN
            used := P01W29_Used;
            subType := P01W29_SubType;
            toolSel := P01W29_ToolSel;
            lenMM := P01W29_LenMM;
            arcStart := P01W29_ArcStart;
            arcEnd := P01W29_ArcEnd;
            approach := P01W29_Approach;
            retract := P01W29_Retract;
            trans := P01W29_Trans;
        ELSEIF slot = 30 THEN
            used := P01W30_Used;
            subType := P01W30_SubType;
            toolSel := P01W30_ToolSel;
            lenMM := P01W30_LenMM;
            arcStart := P01W30_ArcStart;
            arcEnd := P01W30_ArcEnd;
            approach := P01W30_Approach;
            retract := P01W30_Retract;
            trans := P01W30_Trans;
        ELSE
            used := FALSE;
        ENDIF
    ENDPROC

    PROC ClearSlot_P01(num slot)
        IF slot = 1 THEN
            P01W01_Used := FALSE;
            P01W01_SubType := 0;
            P01W01_ToolSel := 0;
            P01W01_LenMM := 0;
            P01W01_ArcStart := [[0,0,0],[1,0,0,0],[0,0,0,0],[9E9,9E9,9E9,9E9,9E9,9E9]];
            P01W01_ArcEnd := [[0,0,0],[1,0,0,0],[0,0,0,0],[9E9,9E9,9E9,9E9,9E9,9E9]];
            P01W01_Approach := [[0,0,0],[1,0,0,0],[0,0,0,0],[9E9,9E9,9E9,9E9,9E9,9E9]];
            P01W01_Retract := [[0,0,0],[1,0,0,0],[0,0,0,0],[9E9,9E9,9E9,9E9,9E9,9E9]];
            P01W01_Trans := [[0,0,0],[1,0,0,0],[0,0,0,0],[9E9,9E9,9E9,9E9,9E9,9E9]];
        ELSEIF slot = 2 THEN
            P01W02_Used := FALSE;
            P01W02_SubType := 0;
            P01W02_ToolSel := 0;
            P01W02_LenMM := 0;
            P01W02_ArcStart := [[0,0,0],[1,0,0,0],[0,0,0,0],[9E9,9E9,9E9,9E9,9E9,9E9]];
            P01W02_ArcEnd := [[0,0,0],[1,0,0,0],[0,0,0,0],[9E9,9E9,9E9,9E9,9E9,9E9]];
            P01W02_Approach := [[0,0,0],[1,0,0,0],[0,0,0,0],[9E9,9E9,9E9,9E9,9E9,9E9]];
            P01W02_Retract := [[0,0,0],[1,0,0,0],[0,0,0,0],[9E9,9E9,9E9,9E9,9E9,9E9]];
            P01W02_Trans := [[0,0,0],[1,0,0,0],[0,0,0,0],[9E9,9E9,9E9,9E9,9E9,9E9]];
        ELSEIF slot = 3 THEN
            P01W03_Used := FALSE;
            P01W03_SubType := 0;
            P01W03_ToolSel := 0;
            P01W03_LenMM := 0;
            P01W03_ArcStart := [[0,0,0],[1,0,0,0],[0,0,0,0],[9E9,9E9,9E9,9E9,9E9,9E9]];
            P01W03_ArcEnd := [[0,0,0],[1,0,0,0],[0,0,0,0],[9E9,9E9,9E9,9E9,9E9,9E9]];
            P01W03_Approach := [[0,0,0],[1,0,0,0],[0,0,0,0],[9E9,9E9,9E9,9E9,9E9,9E9]];
            P01W03_Retract := [[0,0,0],[1,0,0,0],[0,0,0,0],[9E9,9E9,9E9,9E9,9E9,9E9]];
            P01W03_Trans := [[0,0,0],[1,0,0,0],[0,0,0,0],[9E9,9E9,9E9,9E9,9E9,9E9]];
        ELSEIF slot = 4 THEN
            P01W04_Used := FALSE;
            P01W04_SubType := 0;
            P01W04_ToolSel := 0;
            P01W04_LenMM := 0;
            P01W04_ArcStart := [[0,0,0],[1,0,0,0],[0,0,0,0],[9E9,9E9,9E9,9E9,9E9,9E9]];
            P01W04_ArcEnd := [[0,0,0],[1,0,0,0],[0,0,0,0],[9E9,9E9,9E9,9E9,9E9,9E9]];
            P01W04_Approach := [[0,0,0],[1,0,0,0],[0,0,0,0],[9E9,9E9,9E9,9E9,9E9,9E9]];
            P01W04_Retract := [[0,0,0],[1,0,0,0],[0,0,0,0],[9E9,9E9,9E9,9E9,9E9,9E9]];
            P01W04_Trans := [[0,0,0],[1,0,0,0],[0,0,0,0],[9E9,9E9,9E9,9E9,9E9,9E9]];
        ELSEIF slot = 5 THEN
            P01W05_Used := FALSE;
            P01W05_SubType := 0;
            P01W05_ToolSel := 0;
            P01W05_LenMM := 0;
            P01W05_ArcStart := [[0,0,0],[1,0,0,0],[0,0,0,0],[9E9,9E9,9E9,9E9,9E9,9E9]];
            P01W05_ArcEnd := [[0,0,0],[1,0,0,0],[0,0,0,0],[9E9,9E9,9E9,9E9,9E9,9E9]];
            P01W05_Approach := [[0,0,0],[1,0,0,0],[0,0,0,0],[9E9,9E9,9E9,9E9,9E9,9E9]];
            P01W05_Retract := [[0,0,0],[1,0,0,0],[0,0,0,0],[9E9,9E9,9E9,9E9,9E9,9E9]];
            P01W05_Trans := [[0,0,0],[1,0,0,0],[0,0,0,0],[9E9,9E9,9E9,9E9,9E9,9E9]];
        ELSEIF slot = 6 THEN
            P01W06_Used := FALSE;
            P01W06_SubType := 0;
            P01W06_ToolSel := 0;
            P01W06_LenMM := 0;
            P01W06_ArcStart := [[0,0,0],[1,0,0,0],[0,0,0,0],[9E9,9E9,9E9,9E9,9E9,9E9]];
            P01W06_ArcEnd := [[0,0,0],[1,0,0,0],[0,0,0,0],[9E9,9E9,9E9,9E9,9E9,9E9]];
            P01W06_Approach := [[0,0,0],[1,0,0,0],[0,0,0,0],[9E9,9E9,9E9,9E9,9E9,9E9]];
            P01W06_Retract := [[0,0,0],[1,0,0,0],[0,0,0,0],[9E9,9E9,9E9,9E9,9E9,9E9]];
            P01W06_Trans := [[0,0,0],[1,0,0,0],[0,0,0,0],[9E9,9E9,9E9,9E9,9E9,9E9]];
        ELSEIF slot = 7 THEN
            P01W07_Used := FALSE;
            P01W07_SubType := 0;
            P01W07_ToolSel := 0;
            P01W07_LenMM := 0;
            P01W07_ArcStart := [[0,0,0],[1,0,0,0],[0,0,0,0],[9E9,9E9,9E9,9E9,9E9,9E9]];
            P01W07_ArcEnd := [[0,0,0],[1,0,0,0],[0,0,0,0],[9E9,9E9,9E9,9E9,9E9,9E9]];
            P01W07_Approach := [[0,0,0],[1,0,0,0],[0,0,0,0],[9E9,9E9,9E9,9E9,9E9,9E9]];
            P01W07_Retract := [[0,0,0],[1,0,0,0],[0,0,0,0],[9E9,9E9,9E9,9E9,9E9,9E9]];
            P01W07_Trans := [[0,0,0],[1,0,0,0],[0,0,0,0],[9E9,9E9,9E9,9E9,9E9,9E9]];
        ELSEIF slot = 8 THEN
            P01W08_Used := FALSE;
            P01W08_SubType := 0;
            P01W08_ToolSel := 0;
            P01W08_LenMM := 0;
            P01W08_ArcStart := [[0,0,0],[1,0,0,0],[0,0,0,0],[9E9,9E9,9E9,9E9,9E9,9E9]];
            P01W08_ArcEnd := [[0,0,0],[1,0,0,0],[0,0,0,0],[9E9,9E9,9E9,9E9,9E9,9E9]];
            P01W08_Approach := [[0,0,0],[1,0,0,0],[0,0,0,0],[9E9,9E9,9E9,9E9,9E9,9E9]];
            P01W08_Retract := [[0,0,0],[1,0,0,0],[0,0,0,0],[9E9,9E9,9E9,9E9,9E9,9E9]];
            P01W08_Trans := [[0,0,0],[1,0,0,0],[0,0,0,0],[9E9,9E9,9E9,9E9,9E9,9E9]];
        ELSEIF slot = 9 THEN
            P01W09_Used := FALSE;
            P01W09_SubType := 0;
            P01W09_ToolSel := 0;
            P01W09_LenMM := 0;
            P01W09_ArcStart := [[0,0,0],[1,0,0,0],[0,0,0,0],[9E9,9E9,9E9,9E9,9E9,9E9]];
            P01W09_ArcEnd := [[0,0,0],[1,0,0,0],[0,0,0,0],[9E9,9E9,9E9,9E9,9E9,9E9]];
            P01W09_Approach := [[0,0,0],[1,0,0,0],[0,0,0,0],[9E9,9E9,9E9,9E9,9E9,9E9]];
            P01W09_Retract := [[0,0,0],[1,0,0,0],[0,0,0,0],[9E9,9E9,9E9,9E9,9E9,9E9]];
            P01W09_Trans := [[0,0,0],[1,0,0,0],[0,0,0,0],[9E9,9E9,9E9,9E9,9E9,9E9]];
        ELSEIF slot = 10 THEN
            P01W10_Used := FALSE;
            P01W10_SubType := 0;
            P01W10_ToolSel := 0;
            P01W10_LenMM := 0;
            P01W10_ArcStart := [[0,0,0],[1,0,0,0],[0,0,0,0],[9E9,9E9,9E9,9E9,9E9,9E9]];
            P01W10_ArcEnd := [[0,0,0],[1,0,0,0],[0,0,0,0],[9E9,9E9,9E9,9E9,9E9,9E9]];
            P01W10_Approach := [[0,0,0],[1,0,0,0],[0,0,0,0],[9E9,9E9,9E9,9E9,9E9,9E9]];
            P01W10_Retract := [[0,0,0],[1,0,0,0],[0,0,0,0],[9E9,9E9,9E9,9E9,9E9,9E9]];
            P01W10_Trans := [[0,0,0],[1,0,0,0],[0,0,0,0],[9E9,9E9,9E9,9E9,9E9,9E9]];
        ELSEIF slot = 11 THEN
            P01W11_Used := FALSE;
            P01W11_SubType := 0;
            P01W11_ToolSel := 0;
            P01W11_LenMM := 0;
            P01W11_ArcStart := [[0,0,0],[1,0,0,0],[0,0,0,0],[9E9,9E9,9E9,9E9,9E9,9E9]];
            P01W11_ArcEnd := [[0,0,0],[1,0,0,0],[0,0,0,0],[9E9,9E9,9E9,9E9,9E9,9E9]];
            P01W11_Approach := [[0,0,0],[1,0,0,0],[0,0,0,0],[9E9,9E9,9E9,9E9,9E9,9E9]];
            P01W11_Retract := [[0,0,0],[1,0,0,0],[0,0,0,0],[9E9,9E9,9E9,9E9,9E9,9E9]];
            P01W11_Trans := [[0,0,0],[1,0,0,0],[0,0,0,0],[9E9,9E9,9E9,9E9,9E9,9E9]];
        ELSEIF slot = 12 THEN
            P01W12_Used := FALSE;
            P01W12_SubType := 0;
            P01W12_ToolSel := 0;
            P01W12_LenMM := 0;
            P01W12_ArcStart := [[0,0,0],[1,0,0,0],[0,0,0,0],[9E9,9E9,9E9,9E9,9E9,9E9]];
            P01W12_ArcEnd := [[0,0,0],[1,0,0,0],[0,0,0,0],[9E9,9E9,9E9,9E9,9E9,9E9]];
            P01W12_Approach := [[0,0,0],[1,0,0,0],[0,0,0,0],[9E9,9E9,9E9,9E9,9E9,9E9]];
            P01W12_Retract := [[0,0,0],[1,0,0,0],[0,0,0,0],[9E9,9E9,9E9,9E9,9E9,9E9]];
            P01W12_Trans := [[0,0,0],[1,0,0,0],[0,0,0,0],[9E9,9E9,9E9,9E9,9E9,9E9]];
        ELSEIF slot = 13 THEN
            P01W13_Used := FALSE;
            P01W13_SubType := 0;
            P01W13_ToolSel := 0;
            P01W13_LenMM := 0;
            P01W13_ArcStart := [[0,0,0],[1,0,0,0],[0,0,0,0],[9E9,9E9,9E9,9E9,9E9,9E9]];
            P01W13_ArcEnd := [[0,0,0],[1,0,0,0],[0,0,0,0],[9E9,9E9,9E9,9E9,9E9,9E9]];
            P01W13_Approach := [[0,0,0],[1,0,0,0],[0,0,0,0],[9E9,9E9,9E9,9E9,9E9,9E9]];
            P01W13_Retract := [[0,0,0],[1,0,0,0],[0,0,0,0],[9E9,9E9,9E9,9E9,9E9,9E9]];
            P01W13_Trans := [[0,0,0],[1,0,0,0],[0,0,0,0],[9E9,9E9,9E9,9E9,9E9,9E9]];
        ELSEIF slot = 14 THEN
            P01W14_Used := FALSE;
            P01W14_SubType := 0;
            P01W14_ToolSel := 0;
            P01W14_LenMM := 0;
            P01W14_ArcStart := [[0,0,0],[1,0,0,0],[0,0,0,0],[9E9,9E9,9E9,9E9,9E9,9E9]];
            P01W14_ArcEnd := [[0,0,0],[1,0,0,0],[0,0,0,0],[9E9,9E9,9E9,9E9,9E9,9E9]];
            P01W14_Approach := [[0,0,0],[1,0,0,0],[0,0,0,0],[9E9,9E9,9E9,9E9,9E9,9E9]];
            P01W14_Retract := [[0,0,0],[1,0,0,0],[0,0,0,0],[9E9,9E9,9E9,9E9,9E9,9E9]];
            P01W14_Trans := [[0,0,0],[1,0,0,0],[0,0,0,0],[9E9,9E9,9E9,9E9,9E9,9E9]];
        ELSEIF slot = 15 THEN
            P01W15_Used := FALSE;
            P01W15_SubType := 0;
            P01W15_ToolSel := 0;
            P01W15_LenMM := 0;
            P01W15_ArcStart := [[0,0,0],[1,0,0,0],[0,0,0,0],[9E9,9E9,9E9,9E9,9E9,9E9]];
            P01W15_ArcEnd := [[0,0,0],[1,0,0,0],[0,0,0,0],[9E9,9E9,9E9,9E9,9E9,9E9]];
            P01W15_Approach := [[0,0,0],[1,0,0,0],[0,0,0,0],[9E9,9E9,9E9,9E9,9E9,9E9]];
            P01W15_Retract := [[0,0,0],[1,0,0,0],[0,0,0,0],[9E9,9E9,9E9,9E9,9E9,9E9]];
            P01W15_Trans := [[0,0,0],[1,0,0,0],[0,0,0,0],[9E9,9E9,9E9,9E9,9E9,9E9]];
        ELSEIF slot = 16 THEN
            P01W16_Used := FALSE;
            P01W16_SubType := 0;
            P01W16_ToolSel := 0;
            P01W16_LenMM := 0;
            P01W16_ArcStart := [[0,0,0],[1,0,0,0],[0,0,0,0],[9E9,9E9,9E9,9E9,9E9,9E9]];
            P01W16_ArcEnd := [[0,0,0],[1,0,0,0],[0,0,0,0],[9E9,9E9,9E9,9E9,9E9,9E9]];
            P01W16_Approach := [[0,0,0],[1,0,0,0],[0,0,0,0],[9E9,9E9,9E9,9E9,9E9,9E9]];
            P01W16_Retract := [[0,0,0],[1,0,0,0],[0,0,0,0],[9E9,9E9,9E9,9E9,9E9,9E9]];
            P01W16_Trans := [[0,0,0],[1,0,0,0],[0,0,0,0],[9E9,9E9,9E9,9E9,9E9,9E9]];
        ELSEIF slot = 17 THEN
            P01W17_Used := FALSE;
            P01W17_SubType := 0;
            P01W17_ToolSel := 0;
            P01W17_LenMM := 0;
            P01W17_ArcStart := [[0,0,0],[1,0,0,0],[0,0,0,0],[9E9,9E9,9E9,9E9,9E9,9E9]];
            P01W17_ArcEnd := [[0,0,0],[1,0,0,0],[0,0,0,0],[9E9,9E9,9E9,9E9,9E9,9E9]];
            P01W17_Approach := [[0,0,0],[1,0,0,0],[0,0,0,0],[9E9,9E9,9E9,9E9,9E9,9E9]];
            P01W17_Retract := [[0,0,0],[1,0,0,0],[0,0,0,0],[9E9,9E9,9E9,9E9,9E9,9E9]];
            P01W17_Trans := [[0,0,0],[1,0,0,0],[0,0,0,0],[9E9,9E9,9E9,9E9,9E9,9E9]];
        ELSEIF slot = 18 THEN
            P01W18_Used := FALSE;
            P01W18_SubType := 0;
            P01W18_ToolSel := 0;
            P01W18_LenMM := 0;
            P01W18_ArcStart := [[0,0,0],[1,0,0,0],[0,0,0,0],[9E9,9E9,9E9,9E9,9E9,9E9]];
            P01W18_ArcEnd := [[0,0,0],[1,0,0,0],[0,0,0,0],[9E9,9E9,9E9,9E9,9E9,9E9]];
            P01W18_Approach := [[0,0,0],[1,0,0,0],[0,0,0,0],[9E9,9E9,9E9,9E9,9E9,9E9]];
            P01W18_Retract := [[0,0,0],[1,0,0,0],[0,0,0,0],[9E9,9E9,9E9,9E9,9E9,9E9]];
            P01W18_Trans := [[0,0,0],[1,0,0,0],[0,0,0,0],[9E9,9E9,9E9,9E9,9E9,9E9]];
        ELSEIF slot = 19 THEN
            P01W19_Used := FALSE;
            P01W19_SubType := 0;
            P01W19_ToolSel := 0;
            P01W19_LenMM := 0;
            P01W19_ArcStart := [[0,0,0],[1,0,0,0],[0,0,0,0],[9E9,9E9,9E9,9E9,9E9,9E9]];
            P01W19_ArcEnd := [[0,0,0],[1,0,0,0],[0,0,0,0],[9E9,9E9,9E9,9E9,9E9,9E9]];
            P01W19_Approach := [[0,0,0],[1,0,0,0],[0,0,0,0],[9E9,9E9,9E9,9E9,9E9,9E9]];
            P01W19_Retract := [[0,0,0],[1,0,0,0],[0,0,0,0],[9E9,9E9,9E9,9E9,9E9,9E9]];
            P01W19_Trans := [[0,0,0],[1,0,0,0],[0,0,0,0],[9E9,9E9,9E9,9E9,9E9,9E9]];
        ELSEIF slot = 20 THEN
            P01W20_Used := FALSE;
            P01W20_SubType := 0;
            P01W20_ToolSel := 0;
            P01W20_LenMM := 0;
            P01W20_ArcStart := [[0,0,0],[1,0,0,0],[0,0,0,0],[9E9,9E9,9E9,9E9,9E9,9E9]];
            P01W20_ArcEnd := [[0,0,0],[1,0,0,0],[0,0,0,0],[9E9,9E9,9E9,9E9,9E9,9E9]];
            P01W20_Approach := [[0,0,0],[1,0,0,0],[0,0,0,0],[9E9,9E9,9E9,9E9,9E9,9E9]];
            P01W20_Retract := [[0,0,0],[1,0,0,0],[0,0,0,0],[9E9,9E9,9E9,9E9,9E9,9E9]];
            P01W20_Trans := [[0,0,0],[1,0,0,0],[0,0,0,0],[9E9,9E9,9E9,9E9,9E9,9E9]];
        ELSEIF slot = 21 THEN
            P01W21_Used := FALSE;
            P01W21_SubType := 0;
            P01W21_ToolSel := 0;
            P01W21_LenMM := 0;
            P01W21_ArcStart := [[0,0,0],[1,0,0,0],[0,0,0,0],[9E9,9E9,9E9,9E9,9E9,9E9]];
            P01W21_ArcEnd := [[0,0,0],[1,0,0,0],[0,0,0,0],[9E9,9E9,9E9,9E9,9E9,9E9]];
            P01W21_Approach := [[0,0,0],[1,0,0,0],[0,0,0,0],[9E9,9E9,9E9,9E9,9E9,9E9]];
            P01W21_Retract := [[0,0,0],[1,0,0,0],[0,0,0,0],[9E9,9E9,9E9,9E9,9E9,9E9]];
            P01W21_Trans := [[0,0,0],[1,0,0,0],[0,0,0,0],[9E9,9E9,9E9,9E9,9E9,9E9]];
        ELSEIF slot = 22 THEN
            P01W22_Used := FALSE;
            P01W22_SubType := 0;
            P01W22_ToolSel := 0;
            P01W22_LenMM := 0;
            P01W22_ArcStart := [[0,0,0],[1,0,0,0],[0,0,0,0],[9E9,9E9,9E9,9E9,9E9,9E9]];
            P01W22_ArcEnd := [[0,0,0],[1,0,0,0],[0,0,0,0],[9E9,9E9,9E9,9E9,9E9,9E9]];
            P01W22_Approach := [[0,0,0],[1,0,0,0],[0,0,0,0],[9E9,9E9,9E9,9E9,9E9,9E9]];
            P01W22_Retract := [[0,0,0],[1,0,0,0],[0,0,0,0],[9E9,9E9,9E9,9E9,9E9,9E9]];
            P01W22_Trans := [[0,0,0],[1,0,0,0],[0,0,0,0],[9E9,9E9,9E9,9E9,9E9,9E9]];
        ELSEIF slot = 23 THEN
            P01W23_Used := FALSE;
            P01W23_SubType := 0;
            P01W23_ToolSel := 0;
            P01W23_LenMM := 0;
            P01W23_ArcStart := [[0,0,0],[1,0,0,0],[0,0,0,0],[9E9,9E9,9E9,9E9,9E9,9E9]];
            P01W23_ArcEnd := [[0,0,0],[1,0,0,0],[0,0,0,0],[9E9,9E9,9E9,9E9,9E9,9E9]];
            P01W23_Approach := [[0,0,0],[1,0,0,0],[0,0,0,0],[9E9,9E9,9E9,9E9,9E9,9E9]];
            P01W23_Retract := [[0,0,0],[1,0,0,0],[0,0,0,0],[9E9,9E9,9E9,9E9,9E9,9E9]];
            P01W23_Trans := [[0,0,0],[1,0,0,0],[0,0,0,0],[9E9,9E9,9E9,9E9,9E9,9E9]];
        ELSEIF slot = 24 THEN
            P01W24_Used := FALSE;
            P01W24_SubType := 0;
            P01W24_ToolSel := 0;
            P01W24_LenMM := 0;
            P01W24_ArcStart := [[0,0,0],[1,0,0,0],[0,0,0,0],[9E9,9E9,9E9,9E9,9E9,9E9]];
            P01W24_ArcEnd := [[0,0,0],[1,0,0,0],[0,0,0,0],[9E9,9E9,9E9,9E9,9E9,9E9]];
            P01W24_Approach := [[0,0,0],[1,0,0,0],[0,0,0,0],[9E9,9E9,9E9,9E9,9E9,9E9]];
            P01W24_Retract := [[0,0,0],[1,0,0,0],[0,0,0,0],[9E9,9E9,9E9,9E9,9E9,9E9]];
            P01W24_Trans := [[0,0,0],[1,0,0,0],[0,0,0,0],[9E9,9E9,9E9,9E9,9E9,9E9]];
        ELSEIF slot = 25 THEN
            P01W25_Used := FALSE;
            P01W25_SubType := 0;
            P01W25_ToolSel := 0;
            P01W25_LenMM := 0;
            P01W25_ArcStart := [[0,0,0],[1,0,0,0],[0,0,0,0],[9E9,9E9,9E9,9E9,9E9,9E9]];
            P01W25_ArcEnd := [[0,0,0],[1,0,0,0],[0,0,0,0],[9E9,9E9,9E9,9E9,9E9,9E9]];
            P01W25_Approach := [[0,0,0],[1,0,0,0],[0,0,0,0],[9E9,9E9,9E9,9E9,9E9,9E9]];
            P01W25_Retract := [[0,0,0],[1,0,0,0],[0,0,0,0],[9E9,9E9,9E9,9E9,9E9,9E9]];
            P01W25_Trans := [[0,0,0],[1,0,0,0],[0,0,0,0],[9E9,9E9,9E9,9E9,9E9,9E9]];
        ELSEIF slot = 26 THEN
            P01W26_Used := FALSE;
            P01W26_SubType := 0;
            P01W26_ToolSel := 0;
            P01W26_LenMM := 0;
            P01W26_ArcStart := [[0,0,0],[1,0,0,0],[0,0,0,0],[9E9,9E9,9E9,9E9,9E9,9E9]];
            P01W26_ArcEnd := [[0,0,0],[1,0,0,0],[0,0,0,0],[9E9,9E9,9E9,9E9,9E9,9E9]];
            P01W26_Approach := [[0,0,0],[1,0,0,0],[0,0,0,0],[9E9,9E9,9E9,9E9,9E9,9E9]];
            P01W26_Retract := [[0,0,0],[1,0,0,0],[0,0,0,0],[9E9,9E9,9E9,9E9,9E9,9E9]];
            P01W26_Trans := [[0,0,0],[1,0,0,0],[0,0,0,0],[9E9,9E9,9E9,9E9,9E9,9E9]];
        ELSEIF slot = 27 THEN
            P01W27_Used := FALSE;
            P01W27_SubType := 0;
            P01W27_ToolSel := 0;
            P01W27_LenMM := 0;
            P01W27_ArcStart := [[0,0,0],[1,0,0,0],[0,0,0,0],[9E9,9E9,9E9,9E9,9E9,9E9]];
            P01W27_ArcEnd := [[0,0,0],[1,0,0,0],[0,0,0,0],[9E9,9E9,9E9,9E9,9E9,9E9]];
            P01W27_Approach := [[0,0,0],[1,0,0,0],[0,0,0,0],[9E9,9E9,9E9,9E9,9E9,9E9]];
            P01W27_Retract := [[0,0,0],[1,0,0,0],[0,0,0,0],[9E9,9E9,9E9,9E9,9E9,9E9]];
            P01W27_Trans := [[0,0,0],[1,0,0,0],[0,0,0,0],[9E9,9E9,9E9,9E9,9E9,9E9]];
        ELSEIF slot = 28 THEN
            P01W28_Used := FALSE;
            P01W28_SubType := 0;
            P01W28_ToolSel := 0;
            P01W28_LenMM := 0;
            P01W28_ArcStart := [[0,0,0],[1,0,0,0],[0,0,0,0],[9E9,9E9,9E9,9E9,9E9,9E9]];
            P01W28_ArcEnd := [[0,0,0],[1,0,0,0],[0,0,0,0],[9E9,9E9,9E9,9E9,9E9,9E9]];
            P01W28_Approach := [[0,0,0],[1,0,0,0],[0,0,0,0],[9E9,9E9,9E9,9E9,9E9,9E9]];
            P01W28_Retract := [[0,0,0],[1,0,0,0],[0,0,0,0],[9E9,9E9,9E9,9E9,9E9,9E9]];
            P01W28_Trans := [[0,0,0],[1,0,0,0],[0,0,0,0],[9E9,9E9,9E9,9E9,9E9,9E9]];
        ELSEIF slot = 29 THEN
            P01W29_Used := FALSE;
            P01W29_SubType := 0;
            P01W29_ToolSel := 0;
            P01W29_LenMM := 0;
            P01W29_ArcStart := [[0,0,0],[1,0,0,0],[0,0,0,0],[9E9,9E9,9E9,9E9,9E9,9E9]];
            P01W29_ArcEnd := [[0,0,0],[1,0,0,0],[0,0,0,0],[9E9,9E9,9E9,9E9,9E9,9E9]];
            P01W29_Approach := [[0,0,0],[1,0,0,0],[0,0,0,0],[9E9,9E9,9E9,9E9,9E9,9E9]];
            P01W29_Retract := [[0,0,0],[1,0,0,0],[0,0,0,0],[9E9,9E9,9E9,9E9,9E9,9E9]];
            P01W29_Trans := [[0,0,0],[1,0,0,0],[0,0,0,0],[9E9,9E9,9E9,9E9,9E9,9E9]];
        ELSEIF slot = 30 THEN
            P01W30_Used := FALSE;
            P01W30_SubType := 0;
            P01W30_ToolSel := 0;
            P01W30_LenMM := 0;
            P01W30_ArcStart := [[0,0,0],[1,0,0,0],[0,0,0,0],[9E9,9E9,9E9,9E9,9E9,9E9]];
            P01W30_ArcEnd := [[0,0,0],[1,0,0,0],[0,0,0,0],[9E9,9E9,9E9,9E9,9E9,9E9]];
            P01W30_Approach := [[0,0,0],[1,0,0,0],[0,0,0,0],[9E9,9E9,9E9,9E9,9E9,9E9]];
            P01W30_Retract := [[0,0,0],[1,0,0,0],[0,0,0,0],[9E9,9E9,9E9,9E9,9E9,9E9]];
            P01W30_Trans := [[0,0,0],[1,0,0,0],[0,0,0,0],[9E9,9E9,9E9,9E9,9E9,9E9]];
        ELSE
            TPWrite "Invalid weld slot.";
        ENDIF
    ENDPROC

    PROC StoreNextFree_P01(num subType, num toolSel, num lenMM,
                       robtarget arcStart, robtarget arcEnd, robtarget approach, robtarget retract, robtarget trans)
        IF NOT P01W01_Used THEN
            StoreSlot_P01 1, subType, toolSel, lenMM, arcStart, arcEnd, approach, retract, trans;
            nWeldsP01 := nWeldsP01 + 1;
            RETURN;
        ELSEIF NOT P01W02_Used THEN
            StoreSlot_P01 2, subType, toolSel, lenMM, arcStart, arcEnd, approach, retract, trans;
            nWeldsP01 := nWeldsP01 + 1;
            RETURN;
        ELSEIF NOT P01W03_Used THEN
            StoreSlot_P01 3, subType, toolSel, lenMM, arcStart, arcEnd, approach, retract, trans;
            nWeldsP01 := nWeldsP01 + 1;
            RETURN;
        ELSEIF NOT P01W04_Used THEN
            StoreSlot_P01 4, subType, toolSel, lenMM, arcStart, arcEnd, approach, retract, trans;
            nWeldsP01 := nWeldsP01 + 1;
            RETURN;
        ELSEIF NOT P01W05_Used THEN
            StoreSlot_P01 5, subType, toolSel, lenMM, arcStart, arcEnd, approach, retract, trans;
            nWeldsP01 := nWeldsP01 + 1;
            RETURN;
        ELSEIF NOT P01W06_Used THEN
            StoreSlot_P01 6, subType, toolSel, lenMM, arcStart, arcEnd, approach, retract, trans;
            nWeldsP01 := nWeldsP01 + 1;
            RETURN;
        ELSEIF NOT P01W07_Used THEN
            StoreSlot_P01 7, subType, toolSel, lenMM, arcStart, arcEnd, approach, retract, trans;
            nWeldsP01 := nWeldsP01 + 1;
            RETURN;
        ELSEIF NOT P01W08_Used THEN
            StoreSlot_P01 8, subType, toolSel, lenMM, arcStart, arcEnd, approach, retract, trans;
            nWeldsP01 := nWeldsP01 + 1;
            RETURN;
        ELSEIF NOT P01W09_Used THEN
            StoreSlot_P01 9, subType, toolSel, lenMM, arcStart, arcEnd, approach, retract, trans;
            nWeldsP01 := nWeldsP01 + 1;
            RETURN;
        ELSEIF NOT P01W10_Used THEN
            StoreSlot_P01 10, subType, toolSel, lenMM, arcStart, arcEnd, approach, retract, trans;
            nWeldsP01 := nWeldsP01 + 1;
            RETURN;
        ELSEIF NOT P01W11_Used THEN
            StoreSlot_P01 11, subType, toolSel, lenMM, arcStart, arcEnd, approach, retract, trans;
            nWeldsP01 := nWeldsP01 + 1;
            RETURN;
        ELSEIF NOT P01W12_Used THEN
            StoreSlot_P01 12, subType, toolSel, lenMM, arcStart, arcEnd, approach, retract, trans;
            nWeldsP01 := nWeldsP01 + 1;
            RETURN;
        ELSEIF NOT P01W13_Used THEN
            StoreSlot_P01 13, subType, toolSel, lenMM, arcStart, arcEnd, approach, retract, trans;
            nWeldsP01 := nWeldsP01 + 1;
            RETURN;
        ELSEIF NOT P01W14_Used THEN
            StoreSlot_P01 14, subType, toolSel, lenMM, arcStart, arcEnd, approach, retract, trans;
            nWeldsP01 := nWeldsP01 + 1;
            RETURN;
        ELSEIF NOT P01W15_Used THEN
            StoreSlot_P01 15, subType, toolSel, lenMM, arcStart, arcEnd, approach, retract, trans;
            nWeldsP01 := nWeldsP01 + 1;
            RETURN;
        ELSEIF NOT P01W16_Used THEN
            StoreSlot_P01 16, subType, toolSel, lenMM, arcStart, arcEnd, approach, retract, trans;
            nWeldsP01 := nWeldsP01 + 1;
            RETURN;
        ELSEIF NOT P01W17_Used THEN
            StoreSlot_P01 17, subType, toolSel, lenMM, arcStart, arcEnd, approach, retract, trans;
            nWeldsP01 := nWeldsP01 + 1;
            RETURN;
        ELSEIF NOT P01W18_Used THEN
            StoreSlot_P01 18, subType, toolSel, lenMM, arcStart, arcEnd, approach, retract, trans;
            nWeldsP01 := nWeldsP01 + 1;
            RETURN;
        ELSEIF NOT P01W19_Used THEN
            StoreSlot_P01 19, subType, toolSel, lenMM, arcStart, arcEnd, approach, retract, trans;
            nWeldsP01 := nWeldsP01 + 1;
            RETURN;
        ELSEIF NOT P01W20_Used THEN
            StoreSlot_P01 20, subType, toolSel, lenMM, arcStart, arcEnd, approach, retract, trans;
            nWeldsP01 := nWeldsP01 + 1;
            RETURN;
        ELSEIF NOT P01W21_Used THEN
            StoreSlot_P01 21, subType, toolSel, lenMM, arcStart, arcEnd, approach, retract, trans;
            nWeldsP01 := nWeldsP01 + 1;
            RETURN;
        ELSEIF NOT P01W22_Used THEN
            StoreSlot_P01 22, subType, toolSel, lenMM, arcStart, arcEnd, approach, retract, trans;
            nWeldsP01 := nWeldsP01 + 1;
            RETURN;
        ELSEIF NOT P01W23_Used THEN
            StoreSlot_P01 23, subType, toolSel, lenMM, arcStart, arcEnd, approach, retract, trans;
            nWeldsP01 := nWeldsP01 + 1;
            RETURN;
        ELSEIF NOT P01W24_Used THEN
            StoreSlot_P01 24, subType, toolSel, lenMM, arcStart, arcEnd, approach, retract, trans;
            nWeldsP01 := nWeldsP01 + 1;
            RETURN;
        ELSEIF NOT P01W25_Used THEN
            StoreSlot_P01 25, subType, toolSel, lenMM, arcStart, arcEnd, approach, retract, trans;
            nWeldsP01 := nWeldsP01 + 1;
            RETURN;
        ELSEIF NOT P01W26_Used THEN
            StoreSlot_P01 26, subType, toolSel, lenMM, arcStart, arcEnd, approach, retract, trans;
            nWeldsP01 := nWeldsP01 + 1;
            RETURN;
        ELSEIF NOT P01W27_Used THEN
            StoreSlot_P01 27, subType, toolSel, lenMM, arcStart, arcEnd, approach, retract, trans;
            nWeldsP01 := nWeldsP01 + 1;
            RETURN;
        ELSEIF NOT P01W28_Used THEN
            StoreSlot_P01 28, subType, toolSel, lenMM, arcStart, arcEnd, approach, retract, trans;
            nWeldsP01 := nWeldsP01 + 1;
            RETURN;
        ELSEIF NOT P01W29_Used THEN
            StoreSlot_P01 29, subType, toolSel, lenMM, arcStart, arcEnd, approach, retract, trans;
            nWeldsP01 := nWeldsP01 + 1;
            RETURN;
        ELSEIF NOT P01W30_Used THEN
            StoreSlot_P01 30, subType, toolSel, lenMM, arcStart, arcEnd, approach, retract, trans;
            nWeldsP01 := nWeldsP01 + 1;
            RETURN;
        ELSE
            TPWrite "No free weld slots available.";
        ENDIF
    ENDPROC

